C01814=1119.422,-26.499,-49.584,179.647,5.895,149.157
C01815=1119.427,-26.749,-49.572,179.647,5.891,149.156
C01816=1119.432,-26.999,-49.560,179.648,5.887,149.155
C01817=1119.437,-27.248,-49.547,179.648,5.883,149.154
C01818=1119.443,-27.498,-49.535,179.649,5.878,149.153
C01819=1119.448,-27.747,-49.523,179.649,5.874,149.152
C01820=1119.453,-27.997,-49.511,179.649,5.870,149.151
C01821=1119.458,-28.247,-49.498,179.650,5.866,149.150
C01822=1119.463,-28.497,-49.486,179.650,5.862,149.149
C01823=1119.469,-28.746,-49.473,179.651,5.857,149.148
C01824=1119.474,-28.996,-49.461,179.651,5.853,149.147
C01825=1119.479,-29.246,-49.449,179.651,5.850,149.146
C01826=1119.484,-29.495,-49.436,179.652,5.845,149.145
C01827=1119.490,-29.745,-49.424,179.652,5.841,149.144
C01828=1119.495,-29.994,-49.412,179.651,5.837,149.143
C01829=1119.500,-30.244,-49.400,179.652,5.832,149.142
C01830=1119.505,-30.494,-49.387,179.652,5.828,149.141
C01831=1119.511,-30.744,-49.375,179.652,5.824,149.140
C01832=1119.516,-30.993,-49.363,179.652,5.820,149.139
C01833=1119.521,-31.243,-49.351,179.652,5.816,149.138
C01834=1119.526,-31.493,-49.338,179.651,5.811,149.137
C01835=1119.530,-31.742,-49.327,179.652,5.807,149.136
C01836=1119.536,-31.992,-49.314,179.651,5.802,149.135
C01837=1119.541,-32.242,-49.302,179.651,5.798,149.135
C01838=1119.546,-32.491,-49.290,179.651,5.794,149.134
C01839=1119.552,-32.741,-49.278,179.651,5.790,149.133
C01840=1119.556,-32.956,-49.268,179.651,5.786,149.132
C01841=1119.561,-33.171,-49.257,179.650,5.781,149.131
C01842=1119.565,-33.386,-49.247,179.650,5.778,149.130
C01843=1119.570,-33.601,-49.235,179.650,5.774,149.130
C01844=1119.574,-33.816,-49.225,179.650,5.770,149.129
C01845=1119.579,-34.031,-49.215,179.649,5.766,149.128
C01846=1119.583,-34.246,-49.205,179.649,5.762,149.127
C01847=1119.587,-34.462,-49.194,179.648,5.758,149.127
C01848=1119.592,-34.712,-49.183,179.648,5.754,149.126
C01849=1119.598,-34.961,-49.170,179.647,5.749,149.125
C01850=1119.603,-35.211,-49.158,179.647,5.745,149.124
C01851=1119.608,-35.461,-49.146,179.646,5.740,149.123
C01852=1119.613,-35.710,-49.134,179.645,5.735,149.123
C01853=1119.618,-35.960,-49.122,179.645,5.731,149.122
C01854=1119.624,-36.210,-49.110,179.644,5.726,149.121
C01855=1119.629,-36.459,-49.098,179.643,5.722,149.120
C01856=1119.635,-36.708,-49.086,179.643,5.717,149.119
C01857=1119.640,-36.958,-49.075,179.642,5.711,149.118
C01858=1119.645,-37.207,-49.062,179.641,5.707,149.118
C01859=1119.650,-37.457,-49.051,179.640,5.702,149.117
C01860=1119.656,-37.707,-49.039,179.639,5.697,149.116
C01861=1119.660,-37.957,-49.027,179.638,5.692,149.115
C01862=1119.665,-38.206,-49.015,179.637,5.687,149.114
C01863=1119.671,-38.456,-49.003,179.636,5.682,149.114
C01864=1119.676,-38.706,-48.991,179.635,5.677,149.113
C01865=1119.681,-38.955,-48.980,179.635,5.673,149.112
C01866=1119.686,-39.205,-48.968,179.633,5.667,149.111
C01867=1119.691,-39.455,-48.955,179.633,5.663,149.110
C01868=1119.697,-39.705,-48.943,179.631,5.657,149.110
C01869=1119.702,-39.954,-48.932,179.630,5.652,149.109
C01870=1119.708,-40.203,-48.921,179.629,5.646,149.108
C01871=1119.713,-40.453,-48.909,179.628,5.642,149.107
C01872=1119.718,-40.703,-48.897,179.627,5.636,149.106
C01873=1119.723,-40.953,-48.885,179.625,5.631,149.106
C01874=1119.729,-41.203,-48.874,179.624,5.626,149.105
C01875=1119.733,-41.453,-48.862,179.623,5.621,149.104
C01876=1119.738,-41.702,-48.850,179.622,5.615,149.103
C01877=1119.744,-41.951,-48.839,179.621,5.610,149.102
C01878=1119.749,-42.201,-48.827,179.619,5.604,149.102
C01879=1119.755,-42.451,-48.815,179.618,5.598,149.101
C01880=1119.759,-42.700,-48.804,179.616,5.593,149.100
C01881=1119.765,-42.950,-48.792,179.615,5.587,149.099
C01882=1119.770,-43.199,-48.781,179.615,5.583,149.098
C01883=1119.775,-43.449,-48.769,179.615,5.577,149.097
C01884=1119.780,-43.699,-48.758,179.615,5.572,149.096
C01885=1119.785,-43.949,-48.746,179.615,5.568,149.095
C01886=1119.790,-44.198,-48.735,179.615,5.563,149.094
C01887=1119.796,-44.449,-48.723,179.616,5.559,149.093
C01888=1119.802,-44.698,-48.712,179.616,5.554,149.092
C01889=1119.807,-44.948,-48.701,179.615,5.549,149.091
C01890=1119.812,-45.198,-48.689,179.616,5.545,149.090
C01891=1119.817,-45.447,-48.677,179.616,5.539,149.088
C01892=1119.823,-45.696,-48.666,179.617,5.535,149.087
C01893=1119.827,-45.946,-48.655,179.616,5.530,149.086
C01894=1119.833,-46.196,-48.643,179.617,5.526,149.085
C01895=1119.838,-46.446,-48.631,179.617,5.521,149.084
C01896=1119.842,-46.661,-48.622,179.617,5.517,149.083
C01897=1119.847,-46.876,-48.612,179.617,5.513,149.082
C01898=1119.851,-47.091,-48.602,179.617,5.509,149.081
C01899=1119.856,-47.307,-48.592,179.618,5.505,149.080
C01900=1119.861,-47.522,-48.582,179.617,5.500,149.080
C01901=1119.865,-47.737,-48.573,179.617,5.496,149.079
C01902=1119.870,-47.952,-48.563,179.618,5.492,149.078
C01903=1119.874,-48.167,-48.553,179.618,5.489,149.077
C01904=1119.879,-48.417,-48.542,179.618,5.484,149.076
C01905=1119.884,-48.667,-48.530,179.619,5.479,149.075
C01906=1119.890,-48.916,-48.520,179.618,5.474,149.074
C01907=1119.895,-49.166,-48.508,179.619,5.470,149.072
C01908=1119.900,-49.415,-48.496,179.619,5.465,149.071
C01909=1119.906,-49.665,-48.485,179.619,5.461,149.070
C01910=1119.911,-49.915,-48.474,179.619,5.456,149.069
C01911=1119.916,-50.165,-48.463,179.619,5.451,149.068
C01912=1119.921,-50.414,-48.451,179.620,5.446,149.067
C01913=1119.926,-50.663,-48.440,179.619,5.442,149.066
C01914=1119.932,-50.914,-48.429,179.620,5.437,149.065
C01915=1119.937,-51.164,-48.418,179.620,5.432,149.064
C01916=1119.942,-51.412,-48.407,179.620,5.427,149.063
C01917=1119.947,-51.662,-48.395,179.620,5.423,149.062
C01918=1119.952,-51.913,-48.384,179.621,5.418,149.061
C01919=1119.958,-52.162,-48.373,179.621,5.414,149.060
C01920=1119.963,-52.412,-48.361,179.621,5.409,149.058
C01921=1119.968,-52.662,-48.351,179.621,5.404,149.057
C01922=1119.974,-52.911,-48.339,179.621,5.400,149.056
C01923=1119.979,-53.161,-48.328,179.621,5.394,149.055
C01924=1119.984,-53.411,-48.318,179.622,5.390,149.054
C01925=1119.990,-53.660,-48.306,179.622,5.385,149.053
C01926=1119.995,-53.910,-48.295,179.622,5.381,149.052
C01927=1120.000,-54.160,-48.284,179.622,5.376,149.051
C01928=1120.006,-54.409,-48.273,179.622,5.371,149.050
C01929=1120.010,-54.659,-48.261,179.622,5.367,149.049
C01930=1120.015,-54.909,-48.251,179.623,5.362,149.048
C01931=1120.021,-55.158,-48.239,179.623,5.357,149.047
C01932=1120.026,-55.408,-48.228,179.623,5.353,149.046
C01933=1120.031,-55.658,-48.217,179.623,5.347,149.044
C01934=1120.036,-55.907,-48.206,179.623,5.344,149.044
C01935=1120.042,-56.158,-48.195,179.623,5.338,149.042
C01936=1120.047,-56.407,-48.184,179.624,5.334,149.041
C01937=1120.052,-56.656,-48.173,179.624,5.329,149.040
C01938=1120.057,-56.906,-48.163,179.624,5.324,149.039
C01939=1120.063,-57.156,-48.151,179.624,5.320,149.038
C01940=1120.068,-57.406,-48.140,179.624,5.315,149.037
C01941=1120.073,-57.656,-48.129,179.625,5.311,149.036
C01942=1120.078,-57.905,-48.119,179.625,5.306,149.035
C01943=1120.084,-58.155,-48.107,179.625,5.302,149.034
C01944=1120.089,-58.404,-48.096,179.625,5.296,149.033
C01945=1120.094,-58.654,-48.086,179.625,5.291,149.032
C01946=1120.099,-58.904,-48.074,179.625,5.287,149.031
C01947=1120.104,-59.153,-48.064,179.625,5.282,149.029
C01948=1120.110,-59.403,-48.052,179.626,5.278,149.029
C01949=1120.115,-59.653,-48.042,179.626,5.273,149.027
C01950=1120.120,-59.903,-48.031,179.626,5.269,149.026
C01951=1120.125,-60.153,-48.020,179.626,5.264,149.025
C01952=1120.130,-60.368,-48.011,179.626,5.259,149.024
C01953=1120.135,-60.582,-48.001,179.625,5.255,149.024
C01954=1120.139,-60.798,-47.992,179.624,5.251,149.023
C01955=1120.144,-61.013,-47.983,179.623,5.246,149.022
C01956=1120.149,-61.229,-47.973,179.623,5.241,149.021
C01957=1120.152,-61.444,-47.965,179.622,5.237,149.021
C01958=1120.157,-61.659,-47.955,179.622,5.233,149.020
C01959=1120.161,-61.874,-47.945,179.621,5.228,149.019
C01960=1120.167,-62.124,-47.935,179.620,5.223,149.018
C01961=1120.172,-62.374,-47.924,179.620,5.218,149.017
C01962=1120.178,-62.623,-47.913,179.619,5.212,149.016
C01963=1120.183,-62.874,-47.902,179.619,5.208,149.015
C01964=1120.188,-63.123,-47.891,179.618,5.202,149.014
C01965=1120.193,-63.373,-47.881,179.618,5.197,149.013
C01966=1120.199,-63.622,-47.871,179.617,5.191,149.012
C01967=1120.204,-63.872,-47.859,179.617,5.187,149.011
C01968=1120.209,-64.122,-47.849,179.616,5.181,149.010
C01969=1120.214,-64.372,-47.839,179.615,5.176,149.010
C01970=1120.220,-64.621,-47.828,179.615,5.170,149.008
C01971=1120.225,-64.871,-47.817,179.614,5.166,149.007
C01972=1120.230,-65.121,-47.807,179.613,5.160,149.007
C01973=1120.235,-65.371,-47.796,179.613,5.155,149.006
C01974=1120.240,-65.620,-47.785,179.612,5.149,149.004
C01975=1120.245,-65.870,-47.775,179.612,5.145,149.004
C01976=1120.251,-66.119,-47.765,179.611,5.139,149.003
C01977=1120.256,-66.370,-47.754,179.611,5.134,149.001
C01978=1120.262,-66.619,-47.744,179.611,5.129,149.001
C01979=1120.267,-66.868,-47.733,179.610,5.123,148.999
C01980=1120.272,-67.118,-47.722,179.610,5.118,148.998
C01981=1120.278,-67.368,-47.712,179.609,5.113,148.998
C01982=1120.283,-67.618,-47.702,179.609,5.108,148.996
C01983=1120.288,-67.868,-47.691,179.609,5.103,148.995
C01984=1120.293,-68.118,-47.681,179.608,5.097,148.994
C01985=1120.298,-68.367,-47.670,179.608,5.092,148.993
C01986=1120.304,-68.616,-47.660,179.607,5.086,148.992
C01987=1120.309,-68.867,-47.649,179.607,5.081,148.991
C01988=1120.315,-69.116,-47.639,179.607,5.076,148.990
C01989=1120.320,-69.366,-47.629,179.606,5.071,148.989
C01990=1120.325,-69.616,-47.618,179.606,5.066,148.988
C01991=1120.331,-69.866,-47.608,179.607,5.060,148.987
C01992=1120.336,-70.116,-47.597,179.606,5.055,148.986
C01993=1120.341,-70.365,-47.587,179.606,5.050,148.985
C01994=1120.347,-70.615,-47.577,179.605,5.045,148.984
C01995=1120.351,-70.865,-47.567,179.605,5.039,148.983
C01996=1120.357,-71.114,-47.557,179.605,5.034,148.982
C01997=1120.362,-71.364,-47.546,179.605,5.029,148.981
C01998=1120.367,-71.614,-47.536,179.605,5.024,148.979
C01999=1120.373,-71.864,-47.526,179.604,5.018,148.978
C02000=1120.379,-72.113,-47.515,179.604,5.013,148.977
C02001=1120.384,-72.364,-47.505,179.604,5.008,148.976
C02002=1120.389,-72.613,-47.495,179.604,5.002,148.975
C02003=1120.394,-72.862,-47.485,179.604,4.997,148.974
C02004=1120.400,-73.112,-47.475,179.603,4.992,148.973
C02005=1120.405,-73.362,-47.464,179.604,4.987,148.972
C02006=1120.410,-73.612,-47.454,179.604,4.982,148.971
C02007=1120.416,-73.861,-47.444,179.603,4.976,148.970
C02008=1120.420,-74.076,-47.435,179.603,4.972,148.969
C02009=1120.425,-74.292,-47.427,179.603,4.967,148.968
C02010=1120.429,-74.508,-47.418,179.603,4.962,148.967
C02011=1120.434,-74.722,-47.409,179.603,4.958,148.966
C02012=1120.439,-74.939,-47.400,179.603,4.954,148.965
C02013=1120.443,-75.154,-47.392,179.603,4.950,148.964
C02014=1120.448,-75.369,-47.383,179.603,4.945,148.963
C02015=1120.452,-75.584,-47.375,179.603,4.940,148.962
C02016=1120.458,-75.834,-47.365,179.603,4.935,148.961
C02017=1120.463,-76.084,-47.354,179.603,4.929,148.960
C02018=1120.468,-76.333,-47.344,179.603,4.925,148.959
C02019=1120.473,-76.583,-47.334,179.603,4.920,148.957
C02020=1120.479,-76.832,-47.324,179.603,4.914,148.956
C02021=1120.484,-77.083,-47.314,179.603,4.909,148.955
C02022=1120.489,-77.333,-47.305,179.603,4.904,148.954
C02023=1120.495,-77.582,-47.294,179.603,4.899,148.953
C02024=1120.500,-77.832,-47.284,179.603,4.893,148.952
C02025=1120.506,-78.082,-47.275,179.603,4.888,148.950
C02026=1120.510,-78.332,-47.265,179.603,4.883,148.949
C02027=1120.516,-78.581,-47.254,179.603,4.878,148.948
C02028=1120.522,-78.831,-47.244,179.604,4.872,148.947
C02029=1120.527,-79.081,-47.235,179.604,4.867,148.946
C02030=1120.532,-79.330,-47.225,179.604,4.862,148.945
C02031=1120.537,-79.580,-47.215,179.604,4.857,148.943
C02032=1120.542,-79.830,-47.205,179.604,4.852,148.942
C02033=1120.548,-80.080,-47.195,179.604,4.847,148.941
C02034=1120.554,-80.329,-47.185,179.605,4.841,148.940
C02035=1120.559,-80.579,-47.176,179.605,4.836,148.939
C02036=1120.565,-80.829,-47.166,179.605,4.831,148.938
C02037=1120.570,-81.079,-47.156,179.605,4.826,148.936
C02038=1120.574,-81.328,-47.146,179.605,4.821,148.935
C02039=1120.580,-81.578,-47.136,179.605,4.816,148.934
C02040=1120.585,-81.828,-47.127,179.606,4.811,148.933
C02041=1120.591,-82.077,-47.117,179.606,4.806,148.932
C02042=1120.597,-82.327,-47.107,179.606,4.801,148.931
C02043=1120.601,-82.577,-47.097,179.607,4.796,148.929
C02044=1120.607,-82.827,-47.088,179.607,4.791,148.928
C02045=1120.612,-83.077,-47.078,179.607,4.786,148.927
C02046=1120.617,-83.326,-47.068,179.608,4.780,148.926
C02047=1120.622,-83.576,-47.059,179.608,4.775,148.924
C02048=1120.628,-83.826,-47.049,179.608,4.770,148.923
C02049=1120.634,-84.076,-47.039,179.609,4.765,148.922
C02050=1120.639,-84.325,-47.030,179.609,4.760,148.921
C02051=1120.644,-84.575,-47.019,179.609,4.755,148.920
C02052=1120.649,-84.825,-47.010,179.609,4.750,148.919
C02053=1120.655,-85.075,-47.000,179.609,4.745,148.917
C02054=1120.660,-85.324,-46.991,179.611,4.740,148.916
C02055=1120.665,-85.574,-46.981,179.611,4.735,148.915
C02056=1120.670,-85.824,-46.972,179.611,4.730,148.914
C02057=1120.676,-86.073,-46.962,179.611,4.724,148.912
C02058=1120.681,-86.323,-46.953,179.612,4.720,148.911
C02059=1120.687,-86.573,-46.943,179.612,4.715,148.910
C02060=1120.692,-86.823,-46.934,179.612,4.710,148.909
C02061=1120.697,-87.073,-46.923,179.614,4.705,148.907
C02062=1120.702,-87.323,-46.914,179.614,4.700,148.906
C02063=1120.708,-87.572,-46.904,179.614,4.695,148.905
C02064=1120.713,-87.787,-46.896,179.614,4.691,148.904
C02065=1120.717,-88.003,-46.888,179.615,4.686,148.903
C02066=1120.722,-88.218,-46.880,179.615,4.682,148.902
C02067=1120.726,-88.434,-46.872,179.616,4.678,148.901
C02068=1120.730,-88.650,-46.864,179.616,4.673,148.900
C02069=1120.736,-88.865,-46.855,179.617,4.669,148.899
C02070=1120.740,-89.080,-46.847,179.617,4.665,148.898
C02071=1120.745,-89.295,-46.839,179.618,4.661,148.897
C02072=1120.751,-89.545,-46.830,179.618,4.655,148.895
C02073=1120.755,-89.795,-46.820,179.619,4.651,148.894
C02074=1120.760,-90.045,-46.811,179.619,4.646,148.893
C02075=1120.766,-90.295,-46.800,179.620,4.641,148.892
C02076=1120.771,-90.545,-46.792,179.620,4.636,148.890
C02077=1120.777,-90.795,-46.782,179.621,4.632,148.889
C02078=1120.782,-91.044,-46.772,179.621,4.627,148.888
C02079=1120.788,-91.294,-46.763,179.622,4.622,148.887
C02080=1120.793,-91.544,-46.754,179.623,4.617,148.885
C02081=1120.798,-91.793,-46.744,179.624,4.612,148.884
C02082=1120.803,-92.043,-46.735,179.624,4.607,148.883
C02083=1120.809,-92.293,-46.726,179.625,4.603,148.882
C02084=1120.813,-92.543,-46.716,179.625,4.598,148.881
C02085=1120.819,-92.793,-46.707,179.626,4.593,148.879
C02086=1120.825,-93.043,-46.698,179.627,4.589,148.878
C02087=1120.830,-93.292,-46.688,179.627,4.583,148.877
C02088=1120.835,-93.542,-46.679,179.628,4.579,148.876
C02089=1120.840,-93.792,-46.670,179.629,4.573,148.874
C02090=1120.846,-94.041,-46.660,179.629,4.569,148.873
C02091=1120.851,-94.291,-46.651,179.630,4.565,148.872
C02092=1120.856,-94.541,-46.642,179.630,4.560,148.871
C02093=1120.862,-94.791,-46.633,179.630,4.554,148.870
C02094=1120.867,-95.040,-46.623,179.631,4.550,148.868
C02095=1120.872,-95.290,-46.614,179.631,4.545,148.867
C02096=1120.878,-95.540,-46.605,179.632,4.540,148.866
C02097=1120.883,-95.790,-46.595,179.632,4.535,148.865
C02098=1120.889,-96.039,-46.586,179.633,4.530,148.864
C02099=1120.895,-96.289,-46.577,179.633,4.525,148.862
C02100=1120.900,-96.539,-46.568,179.633,4.520,148.862
C02101=1120.905,-96.789,-46.559,179.633,4.515,148.860
C02102=1120.911,-97.038,-46.549,179.634,4.511,148.859
C02103=1120.916,-97.288,-46.540,179.634,4.506,148.858
C02104=1120.921,-97.538,-46.531,179.634,4.500,148.857
C02105=1120.927,-97.788,-46.522,179.634,4.495,148.856
C02106=1120.932,-98.038,-46.513,179.634,4.490,148.854
C02107=1120.937,-98.287,-46.503,179.635,4.486,148.853
C02108=1120.942,-98.537,-46.494,179.635,4.481,148.852
C02109=1120.948,-98.787,-46.485,179.636,4.475,148.851
C02110=1120.953,-99.037,-46.476,179.636,4.470,148.850
C02111=1120.958,-99.287,-46.467,179.636,4.465,148.848
C02112=1120.964,-99.536,-46.458,179.637,4.461,148.847
C02113=1120.970,-99.786,-46.449,179.637,4.456,148.846
C02114=1120.975,-100.035,-46.439,179.637,4.451,148.845
C02115=1120.980,-100.285,-46.430,179.637,4.446,148.844
C02116=1120.985,-100.535,-46.422,179.637,4.441,148.843
C02117=1120.990,-100.785,-46.413,179.638,4.436,148.842
C02118=1120.996,-101.035,-46.403,179.638,4.431,148.840
C02119=1121.001,-101.285,-46.394,179.639,4.426,148.839
C02120=1121.006,-101.500,-46.387,179.639,4.422,148.838
C02121=1121.011,-101.716,-46.379,179.639,4.417,148.837
C02122=1121.015,-101.931,-46.371,179.639,4.413,148.836
C02123=1121.020,-102.146,-46.363,179.640,4.409,148.835
C02124=1121.025,-102.363,-46.356,179.639,4.404,148.834
C02125=1121.029,-102.578,-46.349,179.640,4.400,148.833
C02126=1121.034,-102.793,-46.341,179.641,4.396,148.832
C02127=1121.039,-103.009,-46.332,179.640,4.391,148.831
C02128=1121.044,-103.259,-46.323,179.640,4.386,148.830
C02129=1121.050,-103.509,-46.315,179.641,4.381,148.829
C02130=1121.055,-103.758,-46.306,179.642,4.376,148.827
C02131=1121.060,-104.008,-46.297,179.642,4.371,148.826
C02132=1121.065,-104.258,-46.288,179.642,4.366,148.825
C02133=1121.071,-104.507,-46.279,179.642,4.361,148.824
C02134=1121.076,-104.757,-46.270,179.642,4.355,148.823
C02135=1121.082,-105.007,-46.261,179.643,4.350,148.822
C02136=1121.087,-105.257,-46.252,179.643,4.345,148.820
C02137=1121.092,-105.507,-46.243,179.643,4.340,148.819
C02138=1121.098,-105.756,-46.235,179.643,4.336,148.818
C02139=1121.103,-106.006,-46.226,179.644,4.331,148.817
C02140=1121.108,-106.256,-46.217,179.644,4.326,148.816
C02141=1121.114,-106.506,-46.208,179.644,4.321,148.815
C02142=1121.119,-106.755,-46.199,179.644,4.315,148.813
C02143=1121.125,-107.005,-46.191,179.645,4.310,148.812
C02144=1121.130,-107.255,-46.182,179.645,4.305,148.811
C02145=1121.135,-107.505,-46.173,179.645,4.300,148.810
C02146=1121.140,-107.755,-46.164,179.645,4.295,148.809
C02147=1121.145,-108.005,-46.156,179.646,4.290,148.807
C02148=1121.151,-108.254,-46.147,179.646,4.284,148.806
C02149=1121.157,-108.504,-46.138,179.646,4.279,148.805
C02150=1121.162,-108.754,-46.129,179.646,4.274,148.804
C02151=1121.168,-109.004,-46.120,179.647,4.269,148.803
C02152=1121.173,-109.253,-46.112,179.647,4.264,148.801
C02153=1121.179,-109.503,-46.103,179.647,4.258,148.800
C02154=1121.184,-109.753,-46.094,179.647,4.253,148.799
C02155=1121.189,-110.003,-46.085,179.648,4.248,148.798
C02156=1121.195,-110.253,-46.077,179.648,4.243,148.797
C02157=1121.200,-110.503,-46.069,179.648,4.238,148.795
C02158=1121.205,-110.752,-46.060,179.648,4.233,148.794
C02159=1121.211,-111.002,-46.051,179.649,4.227,148.793
C02160=1121.216,-111.251,-46.042,179.649,4.222,148.792
C02161=1121.221,-111.502,-46.035,179.649,4.217,148.791
C02162=1121.226,-111.751,-46.026,179.649,4.212,148.789
C02163=1121.232,-112.001,-46.017,179.650,4.207,148.788
C02164=1121.237,-112.251,-46.009,179.649,4.202,148.787
C02165=1121.243,-112.501,-46.000,179.650,4.197,148.786
C02166=1121.248,-112.750,-45.992,179.650,4.192,148.785
C02167=1121.254,-113.000,-45.983,179.650,4.186,148.784
C02168=1121.259,-113.250,-45.975,179.650,4.181,148.782
C02169=1121.264,-113.500,-45.966,179.651,4.176,148.781
C02170=1121.270,-113.749,-45.957,179.651,4.171,148.780
C02171=1121.275,-114.000,-45.949,179.652,4.165,148.779
C02172=1121.281,-114.250,-45.940,179.652,4.160,148.777
C02173=1121.286,-114.499,-45.931,179.652,4.155,148.776
C02174=1121.292,-114.749,-45.923,179.653,4.150,148.775
C02175=1121.296,-114.999,-45.915,179.653,4.145,148.774
C02176=1121.301,-115.215,-45.908,179.653,4.140,148.773
C02177=1121.306,-115.430,-45.900,179.653,4.136,148.772
C02178=1121.311,-115.645,-45.894,179.653,4.131,148.771
C02179=1121.316,-115.861,-45.886,179.653,4.127,148.770
C02180=1121.321,-116.077,-45.879,179.653,4.122,148.769
C02181=1121.325,-116.292,-45.872,179.654,4.118,148.768
C02182=1121.329,-116.508,-45.864,179.654,4.113,148.767
C02183=1121.334,-116.723,-45.857,179.654,4.108,148.766
C02184=1121.340,-116.974,-45.849,179.654,4.103,148.764
C02185=1121.345,-117.223,-45.840,179.654,4.098,148.763
C02186=1121.351,-117.473,-45.832,179.655,4.092,148.762
C02187=1121.356,-117.722,-45.824,179.655,4.087,148.761
C02188=1121.361,-117.973,-45.816,179.655,4.082,148.759
C02189=1121.366,-118.223,-45.807,179.656,4.077,148.758
C02190=1121.373,-118.472,-45.799,179.655,4.071,148.757
C02191=1121.378,-118.722,-45.790,179.656,4.066,148.756
C02192=1121.383,-118.972,-45.783,179.656,4.060,148.755
C02193=1121.388,-119.221,-45.774,179.656,4.055,148.753
C02194=1121.394,-119.472,-45.766,179.657,4.050,148.752
C02195=1121.399,-119.721,-45.757,179.657,4.045,148.751
C02196=1121.405,-119.972,-45.749,179.657,4.039,148.750
C02197=1121.410,-120.220,-45.741,179.657,4.034,148.748
C02198=1121.415,-120.471,-45.733,179.658,4.028,148.747
C02199=1121.421,-120.720,-45.725,179.658,4.023,148.746
C02200=1121.427,-120.970,-45.716,179.658,4.018,148.745
C02201=1121.431,-121.220,-45.708,179.658,4.012,148.743
C02202=1121.437,-121.470,-45.700,179.658,4.007,148.742
C02203=1121.443,-121.720,-45.692,179.658,4.001,148.741
C02204=1121.448,-121.969,-45.684,179.659,3.996,148.740
C02205=1121.453,-122.220,-45.676,179.658,3.990,148.739
C02206=1121.459,-122.469,-45.667,179.659,3.985,148.737
C02207=1121.464,-122.719,-45.659,179.660,3.979,148.736
C02208=1121.470,-122.969,-45.652,179.660,3.974,148.735
C02209=1121.475,-123.218,-45.643,179.660,3.968,148.733
C02210=1121.481,-123.468,-45.635,179.660,3.963,148.732
C02211=1121.486,-123.718,-45.628,179.660,3.958,148.731
C02212=1121.491,-123.968,-45.619,179.660,3.953,148.730
C02213=1121.497,-124.218,-45.611,179.661,3.946,148.728
C02214=1121.502,-124.467,-45.604,179.661,3.941,148.727
C02215=1121.507,-124.717,-45.595,179.661,3.936,148.726
C02216=1121.513,-124.967,-45.588,179.661,3.930,148.725
C02217=1121.518,-125.217,-45.579,179.661,3.925,148.724
C02218=1121.524,-125.467,-45.572,179.662,3.919,148.722
C02219=1121.529,-125.717,-45.563,179.662,3.913,148.721
C02220=1121.535,-125.966,-45.555,179.662,3.908,148.720
C02221=1121.540,-126.217,-45.547,179.662,3.903,148.718
C02222=1121.546,-126.466,-45.540,179.662,3.897,148.717
C02223=1121.551,-126.716,-45.531,179.663,3.891,148.716
C02224=1121.556,-126.966,-45.524,179.663,3.886,148.715
C02225=1121.562,-127.215,-45.516,179.663,3.880,148.713
C02226=1121.567,-127.466,-45.509,179.663,3.875,148.712
C02227=1121.573,-127.715,-45.500,179.664,3.870,148.711
C02228=1121.578,-127.965,-45.492,179.664,3.864,148.709
C02229=1121.583,-128.215,-45.485,179.664,3.858,148.708
C02230=1121.589,-128.465,-45.476,179.664,3.852,148.707
C02231=1121.594,-128.715,-45.469,179.665,3.847,148.706
C02232=1121.171,-128.705,-45.495,179.672,3.851,148.704
C02233=1121.166,-128.455,-45.502,179.672,3.857,148.706
C02234=1121.161,-128.205,-45.511,179.672,3.863,148.707
C02235=1121.155,-127.956,-45.519,179.671,3.868,148.708
C02236=1121.150,-127.705,-45.526,179.671,3.873,148.709
C02237=1121.144,-127.456,-45.534,179.671,3.879,148.711
C02238=1121.139,-127.206,-45.541,179.671,3.884,148.712
C02239=1121.133,-126.956,-45.550,179.670,3.890,148.713
C02240=1121.127,-126.707,-45.558,179.670,3.896,148.715
C02241=1121.123,-126.456,-45.566,179.670,3.901,148.716
C02242=1121.117,-126.207,-45.573,179.670,3.906,148.717
C02243=1121.112,-125.957,-45.582,179.669,3.913,148.718
C02244=1121.106,-125.707,-45.590,179.669,3.918,148.720
C02245=1121.101,-125.457,-45.598,179.669,3.923,148.721
C02246=1121.096,-125.208,-45.606,179.669,3.929,148.722
C02247=1121.090,-124.958,-45.614,179.669,3.934,148.723
C02248=1121.084,-124.708,-45.622,179.668,3.940,148.725
C02249=1121.080,-124.458,-45.630,179.668,3.946,148.726
C02250=1121.074,-124.208,-45.638,179.668,3.951,148.727
C02251=1121.068,-123.958,-45.646,179.668,3.956,148.728
C02252=1121.063,-123.709,-45.654,179.667,3.961,148.730
C02253=1121.058,-123.459,-45.662,179.667,3.968,148.731
C02254=1121.051,-123.209,-45.670,179.667,3.973,148.732
C02255=1121.047,-122.959,-45.678,179.666,3.978,148.733
C02256=1121.041,-122.710,-45.686,179.666,3.983,148.735
C02257=1121.035,-122.459,-45.694,179.666,3.989,148.736
C02258=1121.030,-122.210,-45.703,179.666,3.994,148.737
C02259=1121.025,-121.960,-45.710,179.665,4.000,148.739
C02260=1121.020,-121.710,-45.719,179.665,4.005,148.740
C02261=1121.014,-121.460,-45.727,179.665,4.011,148.741
C02262=1121.009,-121.211,-45.735,179.665,4.016,148.742
C02263=1121.003,-120.961,-45.743,179.665,4.022,148.743
C02264=1120.998,-120.711,-45.752,179.665,4.027,148.745
C02265=1120.992,-120.461,-45.760,179.664,4.032,148.746
C02266=1120.987,-120.211,-45.768,179.665,4.038,148.747
C02267=1120.982,-119.961,-45.776,179.664,4.043,148.748
C02268=1120.976,-119.712,-45.784,179.663,4.049,148.750
C02269=1120.971,-119.462,-45.793,179.663,4.054,148.751
C02270=1120.965,-119.212,-45.801,179.663,4.059,148.752
C02271=1120.960,-118.962,-45.809,179.663,4.064,148.753
C02272=1120.955,-118.713,-45.818,179.663,4.070,148.754
C02273=1120.949,-118.463,-45.826,179.663,4.075,148.756
C02274=1120.944,-118.213,-45.835,179.662,4.080,148.757
C02275=1120.938,-117.963,-45.843,179.662,4.086,148.758
C02276=1120.933,-117.714,-45.851,179.662,4.091,148.759
C02277=1120.928,-117.463,-45.859,179.662,4.096,148.761
C02278=1120.922,-117.214,-45.868,179.661,4.101,148.762
C02279=1120.917,-116.963,-45.876,179.662,4.107,148.763
C02280=1120.911,-116.714,-45.884,179.661,4.113,148.764
C02281=1120.907,-116.499,-45.892,179.660,4.117,148.765
C02282=1120.902,-116.283,-45.899,179.661,4.121,148.766
C02283=1120.898,-116.068,-45.906,179.660,4.126,148.767
C02284=1120.893,-115.852,-45.914,179.660,4.131,148.768
C02285=1120.888,-115.637,-45.921,179.660,4.135,148.769
C02286=1120.883,-115.421,-45.928,179.660,4.140,148.771
C02287=1120.879,-115.205,-45.936,179.659,4.144,148.772
C02288=1120.874,-114.989,-45.943,179.659,4.149,148.773
C02289=1120.869,-114.739,-45.952,179.659,4.154,148.774
C02290=1120.863,-114.490,-45.959,179.659,4.159,148.775
C02291=1120.858,-114.240,-45.968,179.659,4.164,148.776
C02292=1120.853,-113.990,-45.977,179.658,4.169,148.777
C02293=1120.847,-113.740,-45.985,179.658,4.174,148.779
C02294=1120.842,-113.491,-45.994,179.658,4.180,148.780
C02295=1120.837,-113.241,-46.003,179.658,4.185,148.781
C02296=1120.831,-112.992,-46.011,179.657,4.190,148.782
C02297=1120.825,-112.741,-46.019,179.658,4.196,148.783
C02298=1120.820,-112.491,-46.028,179.657,4.201,148.785
C02299=1120.815,-112.241,-46.037,179.657,4.206,148.786
C02300=1120.809,-111.992,-46.046,179.657,4.211,148.787
C02301=1120.804,-111.742,-46.054,179.657,4.217,148.788
C02302=1120.799,-111.492,-46.063,179.656,4.222,148.789
C02303=1120.793,-111.243,-46.071,179.656,4.227,148.791
C02304=1120.788,-110.993,-46.080,179.656,4.232,148.792
C02305=1120.782,-110.743,-46.088,179.656,4.237,148.793
C02306=1120.777,-110.493,-46.097,179.655,4.242,148.794
C02307=1120.771,-110.244,-46.106,179.655,4.248,148.795
C02308=1120.766,-109.994,-46.115,179.655,4.253,148.797
C02309=1120.761,-109.744,-46.123,179.655,4.258,148.798
C02310=1120.756,-109.494,-46.132,179.654,4.263,148.799
C02311=1120.750,-109.244,-46.140,179.654,4.268,148.800
C02312=1120.744,-108.994,-46.149,179.653,4.273,148.801
C02313=1120.739,-108.744,-46.158,179.653,4.278,148.803
C02314=1120.734,-108.495,-46.167,179.653,4.283,148.804
C02315=1120.728,-108.246,-46.175,179.653,4.288,148.805
C02316=1120.723,-107.996,-46.184,179.652,4.293,148.806
C02317=1120.718,-107.746,-46.193,179.652,4.298,148.807
C02318=1120.713,-107.496,-46.202,179.652,4.304,148.809
C02319=1120.707,-107.245,-46.210,179.652,4.309,148.810
C02320=1120.702,-106.996,-46.219,179.651,4.314,148.811
C02321=1120.696,-106.746,-46.228,179.651,4.319,148.812
C02322=1120.691,-106.496,-46.237,179.651,4.324,148.813
C02323=1120.685,-106.246,-46.246,179.651,4.329,148.815
C02324=1120.680,-105.997,-46.255,179.650,4.335,148.816
C02325=1120.674,-105.747,-46.264,179.650,4.340,148.817
C02326=1120.669,-105.498,-46.272,179.650,4.345,148.818
C02327=1120.664,-105.248,-46.281,179.649,4.349,148.819
C02328=1120.659,-104.998,-46.290,179.649,4.354,148.821
C02329=1120.654,-104.748,-46.299,179.649,4.359,148.821
C02330=1120.648,-104.498,-46.309,179.649,4.364,148.823
C02331=1120.642,-104.249,-46.317,179.649,4.370,148.824
C02332=1120.637,-103.999,-46.326,179.648,4.375,148.825
C02333=1120.632,-103.749,-46.335,179.648,4.380,148.826
C02334=1120.627,-103.499,-46.344,179.648,4.385,148.827
C02335=1120.621,-103.249,-46.353,179.647,4.389,148.829
C02336=1120.616,-102.999,-46.362,179.647,4.395,148.830
C02337=1120.611,-102.784,-46.369,179.647,4.399,148.831
C02338=1120.607,-102.568,-46.378,179.646,4.404,148.832
C02339=1120.602,-102.353,-46.385,179.646,4.408,148.833
C02340=1120.598,-102.137,-46.393,179.646,4.413,148.834
C02341=1120.593,-101.922,-46.401,179.646,4.416,148.835
C02342=1120.588,-101.706,-46.409,179.645,4.421,148.836
C02343=1120.584,-101.491,-46.417,179.646,4.426,148.837
C02344=1120.579,-101.276,-46.424,179.645,4.430,148.838
C02345=1120.574,-101.026,-46.433,179.645,4.435,148.839
C02346=1120.568,-100.776,-46.443,179.645,4.440,148.840
C02347=1120.563,-100.526,-46.452,179.644,4.444,148.841
C02348=1120.557,-100.277,-46.460,179.644,4.449,148.843
C02349=1120.552,-100.027,-46.469,179.644,4.455,148.844
C02350=1120.547,-99.777,-46.478,179.643,4.460,148.845
C02351=1120.541,-99.527,-46.488,179.643,4.465,148.846
C02352=1120.536,-99.277,-46.497,179.642,4.469,148.847
C02353=1120.531,-99.028,-46.506,179.643,4.474,148.848
C02354=1120.525,-98.777,-46.516,179.642,4.479,148.850
C02355=1120.520,-98.528,-46.524,179.642,4.484,148.851
C02356=1120.514,-98.278,-46.533,179.642,4.490,148.852
C02357=1120.509,-98.029,-46.542,179.641,4.494,148.853
C02358=1120.504,-97.779,-46.552,179.641,4.499,148.854
C02359=1120.498,-97.529,-46.561,179.641,4.504,148.856
C02360=1120.493,-97.279,-46.570,179.640,4.509,148.857
C02361=1120.487,-97.029,-46.580,179.640,4.515,148.858
C02362=1120.482,-96.780,-46.589,179.639,4.519,148.859
C02363=1120.477,-96.530,-46.598,179.639,4.524,148.860
C02364=1120.471,-96.280,-46.608,179.639,4.529,148.861
C02365=1120.466,-96.030,-46.616,179.639,4.534,148.863
C02366=1120.461,-95.781,-46.626,179.638,4.539,148.864
C02367=1120.455,-95.531,-46.636,179.638,4.544,148.865
C02368=1120.450,-95.281,-46.644,179.638,4.549,148.866
C02369=1120.445,-95.031,-46.653,179.638,4.554,148.867
C02370=1120.440,-94.781,-46.664,179.637,4.558,148.868
C02371=1120.434,-94.532,-46.672,179.637,4.563,148.870
C02372=1120.429,-94.282,-46.681,179.637,4.569,148.871
C02373=1120.424,-94.032,-46.692,179.636,4.573,148.872
C02374=1120.418,-93.782,-46.700,179.635,4.578,148.873
C02375=1120.413,-93.532,-46.710,179.634,4.583,148.875
C02376=1120.408,-93.283,-46.720,179.634,4.587,148.876
C02377=1120.403,-93.033,-46.728,179.633,4.592,148.877
C02378=1120.397,-92.783,-46.738,179.632,4.597,148.878
C02379=1120.392,-92.534,-46.748,179.631,4.601,148.879
C02380=1120.387,-92.284,-46.756,179.631,4.607,148.881
C02381=1120.381,-92.034,-46.766,179.630,4.611,148.882
C02382=1120.376,-91.784,-46.776,179.630,4.616,148.883
C02383=1120.370,-91.534,-46.785,179.629,4.621,148.884
C02384=1120.365,-91.285,-46.795,179.629,4.626,148.886
C02385=1120.359,-91.035,-46.804,179.628,4.630,148.887
C02386=1120.354,-90.785,-46.813,179.628,4.635,148.888
C02387=1120.349,-90.536,-46.823,179.627,4.640,148.889
C02388=1120.343,-90.286,-46.832,179.626,4.645,148.891
C02389=1120.338,-90.036,-46.842,179.625,4.650,148.892
C02390=1120.332,-89.786,-46.851,179.625,4.655,148.893
C02391=1120.327,-89.536,-46.860,179.625,4.660,148.894
C02392=1120.322,-89.287,-46.870,179.624,4.664,148.895
C02393=1120.317,-89.071,-46.878,179.624,4.669,148.897
C02394=1120.313,-88.856,-46.886,179.623,4.673,148.897
C02395=1120.308,-88.640,-46.895,179.622,4.677,148.899
C02396=1120.304,-88.425,-46.903,179.623,4.682,148.900
C02397=1120.299,-88.210,-46.911,179.622,4.686,148.901
C02398=1120.295,-87.994,-46.920,179.622,4.690,148.902
C02399=1120.290,-87.779,-46.928,179.621,4.695,148.903
C02400=1120.285,-87.563,-46.936,179.621,4.698,148.904
C02401=1120.280,-87.314,-46.946,179.621,4.704,148.905
C02402=1120.275,-87.064,-46.955,179.620,4.709,148.906
C02403=1120.269,-86.814,-46.965,179.619,4.714,148.908
C02404=1120.264,-86.564,-46.974,179.619,4.719,148.909
C02405=1120.258,-86.315,-46.984,179.619,4.724,148.910
C02406=1120.254,-86.064,-46.993,179.619,4.729,148.911
C02407=1120.248,-85.815,-47.004,179.618,4.733,148.912
C02408=1120.243,-85.566,-47.013,179.618,4.739,148.914
C02409=1120.237,-85.315,-47.023,179.617,4.744,148.915
C02410=1120.232,-85.066,-47.032,179.617,4.749,148.916
C02411=1120.227,-84.816,-47.042,179.616,4.754,148.917
C02412=1120.222,-84.567,-47.051,179.616,4.759,148.918
C02413=1120.216,-84.317,-47.061,179.616,4.764,148.920
C02414=1120.211,-84.067,-47.071,179.615,4.769,148.921
C02415=1120.206,-83.817,-47.081,179.615,4.774,148.922
C02416=1120.200,-83.567,-47.091,179.614,4.779,148.923
C02417=1120.195,-83.318,-47.100,179.614,4.784,148.925
C02418=1120.189,-83.068,-47.110,179.614,4.789,148.926
C02419=1120.184,-82.818,-47.119,179.613,4.794,148.927
C02420=1120.179,-82.569,-47.130,179.613,4.800,148.928
C02421=1120.173,-82.318,-47.139,179.613,4.805,148.929
C02422=1120.169,-82.069,-47.149,179.613,4.810,148.930
C02423=1120.163,-81.819,-47.159,179.613,4.815,148.932
C02424=1120.158,-81.569,-47.168,179.613,4.820,148.933
C02425=1120.152,-81.320,-47.178,179.612,4.825,148.934
C02426=1120.147,-81.070,-47.189,179.612,4.830,148.935
C02427=1120.142,-80.820,-47.198,179.612,4.835,148.936
C02428=1120.136,-80.570,-47.208,179.611,4.840,148.937
C02429=1120.131,-80.321,-47.218,179.611,4.845,148.939
C02430=1120.126,-80.071,-47.228,179.611,4.850,148.940
C02431=1120.120,-79.821,-47.237,179.611,4.855,148.941
C02432=1120.115,-79.571,-47.248,179.611,4.861,148.942
C02433=1120.110,-79.322,-47.258,179.611,4.866,148.943
C02434=1120.104,-79.072,-47.267,179.610,4.871,148.945
C02435=1120.099,-78.822,-47.277,179.610,4.876,148.946
C02436=1120.093,-78.572,-47.287,179.610,4.881,148.947
C02437=1120.089,-78.323,-47.297,179.610,4.886,148.948
C02438=1120.083,-78.073,-47.308,179.610,4.892,148.949
C02439=1120.077,-77.823,-47.317,179.610,4.898,148.950
C02440=1120.073,-77.574,-47.327,179.610,4.903,148.952
C02441=1120.067,-77.324,-47.337,179.610,4.908,148.953
C02442=1120.062,-77.074,-47.348,179.610,4.913,148.954
C02443=1120.056,-76.824,-47.358,179.610,4.918,148.955
C02444=1120.051,-76.574,-47.367,179.609,4.923,148.956
C02445=1120.046,-76.325,-47.377,179.609,4.928,148.957
C02446=1120.041,-76.075,-47.387,179.609,4.934,148.959
C02447=1120.035,-75.825,-47.398,179.609,4.938,148.959
C02448=1120.029,-75.576,-47.408,179.610,4.944,148.961
C02449=1120.025,-75.360,-47.417,179.609,4.949,148.962
C02450=1120.021,-75.144,-47.425,179.610,4.953,148.963
C02451=1120.016,-74.930,-47.433,179.609,4.957,148.964
C02452=1120.011,-74.714,-47.443,179.610,4.962,148.965
C02453=1120.007,-74.498,-47.451,179.610,4.967,148.965
C02454=1120.002,-74.284,-47.460,179.610,4.971,148.966
C02455=1119.998,-74.069,-47.468,179.610,4.976,148.968
C02456=1119.993,-73.853,-47.478,179.609,4.980,148.969
C02457=1119.988,-73.603,-47.488,179.610,4.986,148.969
C02458=1119.983,-73.353,-47.498,179.610,4.991,148.971
C02459=1119.977,-73.104,-47.509,179.610,4.996,148.972
C02460=1119.972,-72.854,-47.518,179.610,5.001,148.973
C02461=1119.966,-72.604,-47.528,179.610,5.006,148.974
C02462=1119.961,-72.354,-47.538,179.611,5.012,148.975
C02463=1119.956,-72.104,-47.549,179.611,5.017,148.976
C02464=1119.950,-71.855,-47.559,179.610,5.022,148.977
C02465=1119.945,-71.605,-47.570,179.611,5.028,148.978
C02466=1119.940,-71.356,-47.580,179.611,5.033,148.979
C02467=1119.934,-71.106,-47.590,179.611,5.038,148.981
C02468=1119.930,-70.856,-47.600,179.612,5.043,148.982
C02469=1119.924,-70.607,-47.611,179.612,5.049,148.983
C02470=1119.919,-70.357,-47.621,179.612,5.053,148.984
C02471=1119.914,-70.107,-47.631,179.612,5.059,148.985
C02472=1119.908,-69.857,-47.642,179.613,5.065,148.986
C02473=1119.903,-69.607,-47.652,179.613,5.069,148.987
C02474=1119.898,-69.358,-47.662,179.613,5.074,148.988
C02475=1119.892,-69.108,-47.673,179.614,5.080,148.989
C02476=1119.887,-68.858,-47.683,179.614,5.085,148.990
C02477=1119.881,-68.608,-47.693,179.614,5.090,148.991
C02478=1119.877,-68.359,-47.705,179.615,5.096,148.992
C02479=1119.871,-68.109,-47.715,179.615,5.101,148.993
C02480=1119.866,-67.860,-47.725,179.615,5.106,148.994
C02481=1119.861,-67.609,-47.736,179.616,5.111,148.995
C02482=1119.855,-67.360,-47.746,179.616,5.116,148.996
C02483=1119.850,-67.110,-47.757,179.617,5.122,148.997
C02484=1119.845,-66.861,-47.767,179.617,5.127,148.998
C02485=1119.840,-66.610,-47.778,179.617,5.132,148.999
C02486=1119.834,-66.361,-47.788,179.617,5.138,149.000
C02487=1119.828,-66.111,-47.798,179.618,5.143,149.001
C02488=1119.824,-65.862,-47.810,179.619,5.148,149.002
C02489=1119.818,-65.612,-47.820,179.619,5.153,149.003
C02490=1119.813,-65.362,-47.830,179.619,5.158,149.004
C02491=1119.808,-65.112,-47.841,179.620,5.164,149.005
C02492=1119.803,-64.863,-47.852,179.620,5.169,149.006
C02493=1119.797,-64.613,-47.862,179.621,5.174,149.007
C02494=1119.792,-64.363,-47.873,179.621,5.179,149.008
C02495=1119.787,-64.114,-47.884,179.622,5.185,149.009
C02496=1119.782,-63.864,-47.894,179.622,5.190,149.010
C02497=1119.776,-63.614,-47.904,179.623,5.195,149.011
C02498=1119.771,-63.364,-47.916,179.623,5.200,149.012
C02499=1119.765,-63.115,-47.927,179.624,5.206,149.013
C02500=1119.760,-62.865,-47.937,179.625,5.211,149.014
C02501=1119.755,-62.616,-47.948,179.626,5.216,149.015
C02502=1119.750,-62.365,-47.959,179.626,5.221,149.016
C02503=1119.745,-62.116,-47.970,179.627,5.227,149.017
C02504=1119.740,-61.866,-47.980,179.627,5.232,149.018
C02505=1119.735,-61.651,-47.989,179.628,5.236,149.019
C02506=1119.731,-61.435,-47.999,179.628,5.241,149.020
C02507=1119.726,-61.220,-48.009,179.629,5.245,149.020
C02508=1119.722,-61.005,-48.018,179.630,5.250,149.021
C02509=1119.717,-60.789,-48.027,179.630,5.254,149.022
C02510=1119.712,-60.575,-48.036,179.631,5.259,149.023
C02511=1119.708,-60.360,-48.046,179.632,5.263,149.023
C02512=1119.703,-60.145,-48.055,179.632,5.267,149.024
C02513=1119.698,-59.895,-48.067,179.632,5.272,149.025
C02514=1119.692,-59.645,-48.077,179.632,5.277,149.026
C02515=1119.688,-59.395,-48.088,179.632,5.281,149.027
C02516=1119.683,-59.145,-48.099,179.632,5.286,149.029
C02517=1119.677,-58.896,-48.110,179.631,5.290,149.029
C02518=1119.672,-58.646,-48.121,179.631,5.295,149.031
C02519=1119.666,-58.397,-48.132,179.631,5.300,149.032
C02520=1119.661,-58.147,-48.142,179.631,5.304,149.033
C02521=1119.657,-57.897,-48.154,179.631,5.310,149.034
C02522=1119.650,-57.647,-48.165,179.630,5.314,149.035
C02523=1119.646,-57.397,-48.176,179.631,5.319,149.036
C02524=1119.641,-57.148,-48.187,179.630,5.323,149.037
C02525=1119.635,-56.898,-48.197,179.630,5.328,149.038
C02526=1119.630,-56.648,-48.209,179.630,5.333,149.039
C02527=1119.624,-56.399,-48.219,179.629,5.337,149.040
C02528=1119.620,-56.149,-48.231,179.630,5.342,149.041
C02529=1119.615,-55.900,-48.242,179.629,5.346,149.042
C02530=1119.609,-55.650,-48.253,179.629,5.352,149.043
C02531=1119.604,-55.400,-48.264,179.629,5.356,149.044
C02532=1119.599,-55.150,-48.275,179.629,5.361,149.046
C02533=1119.593,-54.901,-48.286,179.629,5.366,149.047
C02534=1119.588,-54.651,-48.297,179.629,5.370,149.048
C02535=1119.583,-54.401,-48.308,179.628,5.375,149.049
C02536=1119.577,-54.151,-48.320,179.628,5.379,149.050
C02537=1119.572,-53.902,-48.331,179.628,5.384,149.051
C02538=1119.568,-53.652,-48.342,179.628,5.389,149.052
C02539=1119.561,-53.402,-48.353,179.627,5.393,149.053
C02540=1119.557,-53.153,-48.364,179.628,5.398,149.054
C02541=1119.552,-52.903,-48.376,179.627,5.403,149.055
C02542=1119.546,-52.653,-48.386,179.627,5.408,149.056
C02543=1119.541,-52.404,-48.398,179.627,5.412,149.057
C02544=1119.536,-52.154,-48.409,179.627,5.417,149.058
C02545=1119.530,-51.905,-48.420,179.627,5.422,149.060
C02546=1119.525,-51.654,-48.431,179.626,5.426,149.061
C02547=1119.520,-51.405,-48.443,179.626,5.431,149.062
C02548=1119.515,-51.155,-48.454,179.626,5.436,149.063
C02549=1119.509,-50.906,-48.466,179.626,5.440,149.064
C02550=1119.504,-50.655,-48.476,179.626,5.445,149.065
C02551=1119.499,-50.406,-48.488,179.625,5.450,149.066
C02552=1119.493,-50.157,-48.499,179.625,5.455,149.067
C02553=1119.489,-49.907,-48.510,179.626,5.459,149.068
C02554=1119.483,-49.657,-48.522,179.625,5.464,149.069
C02555=1119.478,-49.407,-48.533,179.625,5.469,149.070
C02556=1119.472,-49.158,-48.544,179.624,5.473,149.071
C02557=1119.468,-48.908,-48.556,179.625,5.478,149.072
C02558=1119.463,-48.658,-48.567,179.624,5.482,149.074
C02559=1119.457,-48.408,-48.579,179.624,5.487,149.075
C02560=1119.452,-48.159,-48.590,179.624,5.492,149.076
C02561=1119.447,-47.944,-48.600,179.624,5.496,149.077
C02562=1119.442,-47.729,-48.610,179.624,5.500,149.077
C02563=1119.438,-47.513,-48.619,179.623,5.504,149.079
C02564=1119.433,-47.298,-48.629,179.623,5.508,149.080
C02565=1119.429,-47.084,-48.639,179.623,5.512,149.080
C02566=1119.425,-46.867,-48.649,179.623,5.516,149.081
C02567=1119.421,-46.652,-48.659,179.623,5.520,149.082
C02568=1119.416,-46.438,-48.669,179.623,5.524,149.083
C02569=1119.410,-46.188,-48.680,179.622,5.529,149.084
C02570=1119.406,-45.939,-48.691,179.623,5.534,149.085
C02571=1119.400,-45.688,-48.703,179.622,5.538,149.086
C02572=1119.395,-45.439,-48.714,179.622,5.544,149.088
C02573=1119.390,-45.189,-48.726,179.621,5.548,149.089
C02574=1119.385,-44.940,-48.737,179.622,5.553,149.090
C02575=1119.379,-44.690,-48.749,179.622,5.558,149.091
C02576=1119.374,-44.440,-48.760,179.621,5.562,149.092
C02577=1119.369,-44.190,-48.772,179.622,5.567,149.093
C02578=1119.364,-43.940,-48.784,179.621,5.571,149.094
C02579=1119.358,-43.691,-48.795,179.621,5.576,149.095
C02580=1119.353,-43.441,-48.806,179.621,5.581,149.096
C02581=1119.348,-43.192,-48.818,179.621,5.585,149.097
C02582=1119.343,-42.942,-48.830,179.621,5.591,149.098
C02583=1119.338,-42.692,-48.841,179.623,5.597,149.099
C02584=1119.332,-42.443,-48.852,179.624,5.602,149.100
C02585=1119.327,-42.193,-48.864,179.625,5.608,149.101
C02586=1119.322,-41.943,-48.876,179.626,5.613,149.101
C02587=1119.316,-41.693,-48.887,179.627,5.618,149.102
C02588=1119.311,-41.444,-48.899,179.629,5.623,149.103
C02589=1119.307,-41.195,-48.911,179.630,5.629,149.104
C02590=1119.301,-40.945,-48.923,179.631,5.634,149.105
C02591=1119.296,-40.695,-48.935,179.633,5.640,149.105
C02592=1119.290,-40.446,-48.946,179.634,5.645,149.106
C02593=1119.285,-40.196,-48.958,179.635,5.650,149.107
C02594=1119.280,-39.946,-48.970,179.636,5.655,149.108
C02595=1119.275,-39.696,-48.981,179.637,5.660,149.109
C02596=1119.270,-39.447,-48.994,179.638,5.666,149.109
C02597=1119.264,-39.197,-49.006,179.639,5.670,149.110
C02598=1119.260,-38.947,-49.017,179.640,5.676,149.111
C02599=1119.254,-38.697,-49.029,179.642,5.681,149.112
C02600=1119.249,-38.447,-49.041,179.642,5.686,149.113
C02601=1119.244,-38.198,-49.053,179.644,5.691,149.113
C02602=1119.239,-37.949,-49.065,179.644,5.696,149.114
C02603=1119.233,-37.699,-49.076,179.644,5.700,149.115
C02604=1119.228,-37.449,-49.088,179.646,5.705,149.116
C02605=1119.222,-37.200,-49.101,179.646,5.710,149.117
C02606=1119.217,-36.950,-49.112,179.647,5.715,149.117
C02607=1119.212,-36.701,-49.124,179.648,5.719,149.118
C02608=1119.207,-36.451,-49.136,179.649,5.725,149.119
C02609=1119.202,-36.201,-49.148,179.650,5.729,149.120
C02610=1119.196,-35.951,-49.160,179.650,5.734,149.121
C02611=1119.191,-35.702,-49.173,179.651,5.739,149.122
C02612=1119.187,-35.452,-49.184,179.652,5.743,149.122
C02613=1119.181,-35.202,-49.196,179.652,5.748,149.123
C02614=1119.176,-34.953,-49.208,179.653,5.753,149.124
C02615=1119.171,-34.703,-49.220,179.653,5.757,149.125
C02616=1119.165,-34.454,-49.233,179.654,5.762,149.126
C02617=1119.161,-34.239,-49.243,179.654,5.766,149.127
C02618=1119.157,-34.023,-49.254,179.654,5.769,149.127
C02619=1119.152,-33.808,-49.264,179.655,5.773,149.128
C02620=1119.148,-33.593,-49.274,179.655,5.777,149.129
C02621=1119.143,-33.378,-49.285,179.655,5.781,149.130
C02622=1119.139,-33.163,-49.295,179.656,5.785,149.130
C02623=1119.134,-32.948,-49.306,179.656,5.788,149.131
C02624=1119.130,-32.733,-49.316,179.656,5.792,149.132
C02625=1119.125,-32.483,-49.328,179.656,5.797,149.133
C02626=1119.119,-32.234,-49.341,179.657,5.802,149.134
C02627=1119.114,-31.984,-49.353,179.657,5.805,149.134
C02628=1119.109,-31.735,-49.365,179.657,5.810,149.135
C02629=1119.103,-31.485,-49.377,179.657,5.814,149.136
C02630=1119.098,-31.235,-49.390,179.657,5.819,149.137
C02631=1119.093,-30.986,-49.402,179.657,5.823,149.138
C02632=1119.089,-30.736,-49.414,179.657,5.827,149.139
C02633=1119.084,-30.486,-49.426,179.658,5.831,149.140
C02634=1119.079,-30.237,-49.438,179.657,5.835,149.141
C02635=1119.073,-29.987,-49.450,179.657,5.840,149.142
C02636=1119.068,-29.737,-49.463,179.657,5.844,149.143
C02637=1119.063,-29.487,-49.475,179.657,5.848,149.144
C02638=1119.057,-29.238,-49.487,179.656,5.853,149.145
C02639=1119.052,-28.989,-49.500,179.656,5.857,149.146
C02640=1119.047,-28.739,-49.512,179.656,5.861,149.147
C02641=1119.042,-28.489,-49.524,179.656,5.865,149.148
C02642=1119.036,-28.240,-49.536,179.655,5.869,149.149
C02643=1119.032,-27.990,-49.549,179.655,5.873,149.150
C02644=1119.027,-27.740,-49.562,179.655,5.878,149.151
C02645=1119.021,-27.490,-49.574,179.655,5.882,149.152
C02646=1119.016,-27.241,-49.586,179.653,5.886,149.153
C02647=1119.011,-26.991,-49.598,179.653,5.890,149.154
C02648=1119.006,-26.742,-49.611,179.653,5.894,149.155
C02649=1119.000,-26.492,-49.624,179.652,5.898,149.156
C02650=1118.995,-26.242,-49.635,179.651,5.903,149.157
C02651=1118.991,-25.992,-49.648,179.651,5.907,149.158
C02652=1118.985,-25.743,-49.661,179.651,5.911,149.159
C02653=1118.980,-25.493,-49.673,179.652,5.917,149.160
C02654=1118.975,-25.244,-49.685,179.652,5.921,149.161
C02655=1118.970,-24.995,-49.698,179.653,5.926,149.162
C02656=1118.964,-24.745,-49.710,179.653,5.931,149.163
C02657=1118.959,-24.495,-49.723,179.654,5.935,149.164
C02658=1118.955,-24.245,-49.736,179.655,5.941,149.165
C02659=1118.949,-23.995,-49.747,179.655,5.946,149.166
C02660=1118.943,-23.746,-49.761,179.656,5.950,149.167
C02661=1118.938,-23.496,-49.773,179.656,5.955,149.167
C02662=1118.933,-23.246,-49.785,179.657,5.960,149.168
C02663=1118.928,-22.997,-49.798,179.658,5.964,149.169
C02664=1118.923,-22.747,-49.811,179.659,5.970,149.170
C02665=1118.918,-22.498,-49.823,179.659,5.975,149.171
C02666=1118.913,-22.248,-49.836,179.660,5.979,149.172
C02667=1118.907,-21.999,-49.848,179.660,5.984,149.173
C02668=1118.902,-21.749,-49.861,179.661,5.989,149.173
C02669=1118.897,-21.499,-49.874,179.661,5.994,149.174
C02670=1118.892,-21.250,-49.886,179.662,5.998,149.175
C02671=1118.887,-21.000,-49.899,179.663,6.003,149.176
C02672=1118.881,-20.750,-49.911,179.663,6.007,149.177
C02673=1118.877,-20.535,-49.923,179.664,6.012,149.178
C02674=1118.872,-20.320,-49.934,179.665,6.016,149.178
C02675=1118.868,-20.106,-49.944,179.665,6.020,149.179
C02676=1118.864,-19.890,-49.956,179.665,6.025,149.180
C02677=1118.859,-19.675,-49.966,179.666,6.028,149.181
C02678=1118.855,-19.461,-49.977,179.667,6.033,149.181
C02679=1118.850,-19.245,-49.988,179.667,6.036,149.182
C02680=1118.846,-19.030,-49.999,179.668,6.041,149.183
C02681=1118.840,-18.781,-50.012,179.668,6.046,149.184
C02682=1118.836,-18.531,-50.025,179.669,6.050,149.184
C02683=1118.831,-18.282,-50.037,179.669,6.055,149.185
C02684=1118.825,-18.032,-50.051,179.670,6.059,149.186
C02685=1118.820,-17.782,-50.064,179.670,6.064,149.187
C02686=1118.815,-17.533,-50.076,179.671,6.068,149.188
C02687=1118.810,-17.284,-50.089,179.672,6.073,149.189
C02688=1118.804,-17.034,-50.102,179.672,6.078,149.190
C02689=1118.800,-16.784,-50.115,179.673,6.083,149.190
C02690=1118.795,-16.535,-50.128,179.673,6.087,149.191
C02691=1118.790,-16.285,-50.140,179.674,6.092,149.192
C02692=1118.784,-16.035,-50.154,179.675,6.096,149.193
C02693=1118.779,-15.786,-50.166,179.675,6.101,149.194
C02694=1118.774,-15.536,-50.179,179.676,6.106,149.195
C02695=1118.769,-15.286,-50.192,179.677,6.110,149.195
C02696=1118.764,-15.037,-50.205,179.677,6.115,149.196
C02697=1118.759,-14.787,-50.218,179.678,6.120,149.197
C02698=1118.753,-14.537,-50.231,179.678,6.124,149.198
C02699=1118.748,-14.288,-50.244,179.679,6.129,149.199
C02700=1118.743,-14.038,-50.256,179.680,6.134,149.200
C02701=1118.738,-13.788,-50.270,179.680,6.138,149.200
C02702=1118.733,-13.539,-50.283,179.681,6.143,149.201
C02703=1118.728,-13.290,-50.296,179.682,6.147,149.202
C02704=1118.723,-13.040,-50.309,179.682,6.152,149.203
C02705=1118.717,-12.790,-50.322,179.683,6.157,149.204
C02706=1118.712,-12.540,-50.336,179.684,6.161,149.205
C02707=1118.707,-12.291,-50.348,179.684,6.166,149.205
C02708=1118.702,-12.042,-50.362,179.685,6.171,149.206
C02709=1118.697,-11.792,-50.375,179.685,6.175,149.207
C02710=1118.692,-11.542,-50.388,179.686,6.180,149.208
C02711=1118.687,-11.292,-50.401,179.687,6.184,149.209
C02712=1118.681,-11.043,-50.414,179.687,6.189,149.210
C02713=1118.677,-10.794,-50.427,179.688,6.193,149.210
C02714=1118.671,-10.544,-50.441,179.689,6.198,149.211
C02715=1118.666,-10.294,-50.453,179.689,6.203,149.212
C02716=1118.661,-10.044,-50.467,179.690,6.207,149.213
C02717=1118.656,-9.795,-50.480,179.691,6.212,149.214
C02718=1118.651,-9.545,-50.494,179.691,6.217,149.215
C02719=1118.646,-9.296,-50.506,179.692,6.221,149.215
C02720=1118.640,-9.046,-50.520,179.693,6.226,149.216
C02721=1118.636,-8.797,-50.533,179.693,6.230,149.217
C02722=1118.630,-8.547,-50.546,179.694,6.235,149.218
C02723=1118.625,-8.297,-50.559,179.694,6.239,149.219
C02724=1118.620,-8.048,-50.573,179.695,6.243,149.219
C02725=1118.615,-7.798,-50.586,179.695,6.248,149.220
C02726=1118.609,-7.548,-50.600,179.696,6.253,149.221
C02727=1118.605,-7.299,-50.613,179.697,6.257,149.222
C02728=1118.599,-7.049,-50.626,179.697,6.262,149.223
C02729=1118.595,-6.834,-50.638,179.698,6.266,149.223
C02730=1118.590,-6.620,-50.649,179.699,6.270,149.224
C02731=1118.586,-6.404,-50.661,179.699,6.273,149.225
C02732=1118.581,-6.190,-50.672,179.699,6.278,149.226
C02733=1118.577,-5.974,-50.684,179.700,6.282,149.226
C02734=1118.573,-5.761,-50.696,179.700,6.285,149.227
C02735=1118.569,-5.545,-50.708,179.701,6.290,149.228
C02736=1118.564,-5.331,-50.719,179.702,6.293,149.228
C02737=1118.559,-5.081,-50.732,179.702,6.298,149.229
C02738=1118.554,-4.832,-50.746,179.703,6.303,149.230
C02739=1118.549,-4.582,-50.759,179.704,6.307,149.231
C02740=1118.544,-4.332,-50.773,179.704,6.312,149.232
C02741=1118.538,-4.082,-50.786,179.705,6.316,149.232
C02742=1118.534,-3.833,-50.800,179.705,6.320,149.233
C02743=1118.528,-3.583,-50.813,179.706,6.325,149.234
C02744=1118.523,-3.334,-50.828,179.706,6.329,149.235
C02745=1118.518,-3.084,-50.840,179.707,6.334,149.236
C02746=1118.513,-2.835,-50.854,179.708,6.338,149.236
C02747=1118.508,-2.585,-50.867,179.708,6.343,149.237
C02748=1118.503,-2.336,-50.881,179.709,6.348,149.238
C02749=1118.497,-2.086,-50.895,179.710,6.352,149.239
C02750=1118.492,-1.836,-50.909,179.710,6.357,149.240
C02751=1118.488,-1.586,-50.922,179.710,6.361,149.241
C02752=1118.482,-1.337,-50.936,179.711,6.365,149.242
C02753=1118.477,-1.087,-50.950,179.712,6.370,149.242
C02754=1118.472,-0.838,-50.963,179.712,6.375,149.243
C02755=1118.467,-0.588,-50.977,179.713,6.379,149.244
C02756=1118.462,-0.339,-50.991,179.714,6.384,149.245
C02757=1118.457,-0.089,-51.004,179.714,6.388,149.246
C02758=1118.452,0.160,-51.018,179.715,6.393,149.246
C02759=1118.446,0.410,-51.031,179.715,6.397,149.247
C02760=1118.441,0.660,-51.045,179.716,6.401,149.248
C02761=1118.437,0.909,-51.059,179.716,6.406,149.249
C02762=1118.431,1.159,-51.072,179.717,6.411,149.250
C02763=1118.426,1.408,-51.087,179.717,6.415,149.251
C02764=1118.421,1.658,-51.101,179.718,6.420,149.251
C02765=1118.416,1.907,-51.115,179.719,6.425,149.252
C02766=1118.411,2.157,-51.128,179.719,6.428,149.253
C02767=1118.406,2.406,-51.142,179.719,6.433,149.254
C02768=1118.401,2.656,-51.156,179.720,6.437,149.255
C02769=1118.396,2.906,-51.170,179.721,6.442,149.256
C02770=1118.391,3.155,-51.183,179.721,6.447,149.256
C02771=1118.386,3.405,-51.197,179.722,6.452,149.257
C02772=1118.381,3.654,-51.211,179.722,6.456,149.258
C02773=1118.375,3.903,-51.225,179.723,6.461,149.259
C02774=1118.370,4.154,-51.239,179.723,6.465,149.260
C02775=1118.365,4.403,-51.253,179.724,6.469,149.261
C02776=1118.360,4.652,-51.266,179.724,6.474,149.261
C02777=1118.355,4.902,-51.281,179.725,6.479,149.262
C02778=1118.350,5.151,-51.295,179.726,6.483,149.263
C02779=1118.345,5.401,-51.309,179.727,6.488,149.264
C02780=1118.340,5.651,-51.323,179.727,6.493,149.265
C02781=1118.335,5.901,-51.337,179.727,6.496,149.266
C02782=1118.330,6.150,-51.351,179.728,6.501,149.267
C02783=1118.324,6.399,-51.365,179.728,6.506,149.267
C02784=1118.320,6.649,-51.379,179.729,6.510,149.268
C02785=1118.315,6.864,-51.391,179.729,6.514,149.269
C02786=1118.311,7.079,-51.403,179.730,6.518,149.270
C02787=1118.306,7.293,-51.415,179.730,6.522,149.270
C02788=1118.303,7.508,-51.427,179.730,6.526,149.271
C02789=1118.298,7.723,-51.440,179.731,6.530,149.272
C02790=1118.293,7.938,-51.451,179.732,6.534,149.273
C02791=1118.289,8.152,-51.464,179.732,6.538,149.273
C02792=1118.284,8.368,-51.476,179.733,6.542,149.274
C02793=1118.279,8.617,-51.490,179.733,6.547,149.275
C02794=1118.275,8.866,-51.504,179.734,6.551,149.276
C02795=1118.270,9.116,-51.518,179.734,6.556,149.277
C02796=1118.265,9.366,-51.532,179.735,6.560,149.277
C02797=1118.260,9.615,-51.546,179.736,6.565,149.278
C02798=1118.254,9.864,-51.560,179.737,6.570,149.279
C02799=1118.249,10.114,-51.575,179.737,6.575,149.280
C02800=1118.244,10.364,-51.589,179.738,6.579,149.281
C02801=1118.239,10.613,-51.603,179.739,6.584,149.282
C02802=1118.234,10.863,-51.617,179.739,6.588,149.282
C02803=1118.229,11.112,-51.631,179.740,6.593,149.283
C02804=1118.224,11.362,-51.646,179.741,6.597,149.284
C02805=1118.218,11.612,-51.661,179.741,6.602,149.285
C02806=1118.214,11.861,-51.676,179.742,6.606,149.285
C02807=1118.209,12.111,-51.690,179.743,6.611,149.286
C02808=1118.203,12.360,-51.704,179.743,6.616,149.287
C02809=1118.198,12.609,-51.718,179.745,6.620,149.288
C02810=1118.193,12.859,-51.732,179.745,6.625,149.289
C02811=1118.188,13.109,-51.747,179.746,6.630,149.290
C02812=1118.183,13.359,-51.761,179.747,6.634,149.290
C02813=1118.178,13.608,-51.775,179.747,6.639,149.291
C02814=1118.174,13.857,-51.790,179.748,6.643,149.292
C02815=1118.168,14.106,-51.804,179.749,6.648,149.293
C02816=1118.163,14.356,-51.818,179.749,6.652,149.294
C02817=1118.158,14.606,-51.833,179.750,6.657,149.294
C02818=1118.152,14.856,-51.847,179.751,6.661,149.295
C02819=1118.148,15.105,-51.862,179.751,6.665,149.296
C02820=1118.143,15.355,-51.877,179.752,6.670,149.297
C02821=1118.138,15.604,-51.891,179.753,6.674,149.297
C02822=1118.133,15.854,-51.905,179.754,6.679,149.298
C02823=1118.128,16.102,-51.920,179.755,6.683,149.299
C02824=1118.123,16.352,-51.934,179.755,6.688,149.300
C02825=1118.117,16.602,-51.949,179.756,6.692,149.301
C02826=1118.112,16.852,-51.963,179.757,6.697,149.301
C02827=1118.107,17.101,-51.978,179.758,6.701,149.302
C02828=1118.102,17.351,-51.993,179.758,6.706,149.303
C02829=1118.097,17.600,-52.007,179.759,6.710,149.303
C02830=1118.092,17.850,-52.022,179.760,6.715,149.304
C02831=1118.087,18.099,-52.037,179.761,6.719,149.305
C02832=1118.082,18.349,-52.051,179.762,6.724,149.306
C02833=1118.078,18.598,-52.066,179.763,6.728,149.307
C02834=1118.072,18.848,-52.081,179.763,6.733,149.307
C02835=1118.067,19.098,-52.095,179.764,6.737,149.308
C02836=1118.062,19.346,-52.110,179.765,6.741,149.309
C02837=1118.057,19.596,-52.124,179.766,6.746,149.310
C02838=1118.051,19.846,-52.140,179.767,6.751,149.310
C02839=1118.046,20.095,-52.154,179.767,6.755,149.311
C02840=1118.042,20.344,-52.169,179.768,6.760,149.312
C02841=1118.037,20.559,-52.182,179.769,6.763,149.312
C02842=1118.033,20.774,-52.194,179.769,6.767,149.313
C02843=1118.029,20.989,-52.207,179.770,6.771,149.314
C02844=1118.025,21.204,-52.220,179.771,6.774,149.314
C02845=1118.020,21.418,-52.233,179.772,6.779,149.315
C02846=1118.016,21.633,-52.245,179.773,6.782,149.316
C02847=1118.012,21.848,-52.258,179.773,6.785,149.316
C02848=1118.007,22.062,-52.271,179.774,6.790,149.317
C02849=1118.002,22.312,-52.285,179.775,6.794,149.317
C02850=1117.997,22.561,-52.300,179.776,6.799,149.318
C02851=1117.992,22.812,-52.315,179.777,6.803,149.319
C02852=1117.987,23.061,-52.330,179.778,6.807,149.320
C02853=1117.982,23.311,-52.344,179.778,6.812,149.321
C02854=1117.977,23.560,-52.360,179.779,6.816,149.321
C02855=1117.972,23.809,-52.375,179.780,6.820,149.322
C02856=1117.967,24.059,-52.389,179.781,6.824,149.322
C02857=1117.962,24.308,-52.405,179.782,6.829,149.323
C02858=1117.957,24.558,-52.419,179.783,6.833,149.324
C02859=1117.951,24.807,-52.435,179.784,6.838,149.325
C02860=1117.947,25.056,-52.450,179.785,6.842,149.325
C02861=1117.942,25.306,-52.464,179.785,6.847,149.326
C02862=1117.936,25.556,-52.480,179.786,6.851,149.327
C02863=1117.932,25.805,-52.494,179.787,6.855,149.328
C02864=1117.926,26.055,-52.509,179.788,6.860,149.328
C02865=1117.922,26.304,-52.524,179.789,6.864,149.329
C02866=1117.916,26.554,-52.539,179.790,6.869,149.330
C02867=1117.911,26.803,-52.554,179.791,6.872,149.330
C02868=1117.906,27.053,-52.570,179.792,6.876,149.331
C02869=1117.902,27.302,-52.585,179.793,6.881,149.332
C02870=1117.896,27.552,-52.600,179.794,6.885,149.332
C02871=1117.891,27.801,-52.615,179.795,6.889,149.333
C02872=1117.886,28.051,-52.631,179.795,6.894,149.334
C02873=1117.881,28.300,-52.645,179.796,6.898,149.334
C02874=1117.876,28.550,-52.661,179.797,6.903,149.335
C02875=1117.871,28.799,-52.676,179.798,6.907,149.336
C02876=1117.866,29.049,-52.692,179.800,6.911,149.336
C02877=1117.862,29.298,-52.707,179.801,6.916,149.337
C02878=1117.856,29.548,-52.721,179.802,6.920,149.338
C02879=1117.851,29.797,-52.736,179.802,6.923,149.338
C02880=1117.846,30.046,-52.752,179.803,6.928,149.339
C02881=1117.841,30.296,-52.767,179.804,6.932,149.340
C02882=1117.836,30.545,-52.783,179.805,6.937,149.341
C02883=1117.831,30.795,-52.797,179.806,6.941,149.341
C02884=1117.826,31.045,-52.813,179.807,6.945,149.342
C02885=1117.821,31.294,-52.828,179.808,6.950,149.343
C02886=1117.816,31.543,-52.843,179.809,6.954,149.343
C02887=1117.811,31.793,-52.859,179.810,6.958,149.344
C02888=1117.807,32.042,-52.874,179.811,6.963,149.344
C02889=1117.801,32.292,-52.890,179.812,6.966,149.345
C02890=1117.796,32.541,-52.906,179.813,6.970,149.346
C02891=1117.791,32.790,-52.921,179.814,6.975,149.346
C02892=1117.786,33.040,-52.936,179.815,6.979,149.347
C02893=1117.781,33.290,-52.951,179.816,6.983,149.348
C02894=1117.776,33.540,-52.966,179.817,6.988,149.348
C02895=1117.771,33.789,-52.982,179.818,6.992,149.349
C02896=1117.766,34.038,-52.997,179.819,6.996,149.350
C02897=1117.762,34.252,-53.011,179.820,6.999,149.350
C02898=1117.757,34.467,-53.024,179.820,7.003,149.351
C02899=1117.753,34.682,-53.037,179.821,7.007,149.351
C02900=1117.749,34.896,-53.051,179.822,7.010,149.352
C02901=1117.745,35.112,-53.064,179.823,7.015,149.353
C02902=1117.740,35.326,-53.078,179.824,7.018,149.353
C02903=1117.736,35.541,-53.091,179.825,7.021,149.354
C02904=1117.732,35.755,-53.104,179.826,7.025,149.354
C02905=1117.727,36.004,-53.120,179.827,7.029,149.355
C02906=1117.721,36.254,-53.135,179.828,7.033,149.355
C02907=1117.717,36.504,-53.151,179.829,7.037,149.356
C02908=1117.712,36.753,-53.166,179.830,7.042,149.357
C02909=1117.706,37.002,-53.182,179.831,7.046,149.357
C02910=1117.701,37.252,-53.197,179.832,7.050,149.358
C02911=1117.696,37.502,-53.213,179.833,7.055,149.359
C02912=1117.692,37.750,-53.229,179.835,7.059,149.359
C02913=1117.687,38.000,-53.245,179.836,7.063,149.360
C02914=1117.682,38.250,-53.261,179.836,7.066,149.360
C02915=1117.676,38.499,-53.276,179.837,7.071,149.361
C02916=1117.671,38.749,-53.292,179.838,7.075,149.362
C02917=1117.667,38.998,-53.307,179.839,7.079,149.362
C02918=1117.662,39.248,-53.323,179.841,7.084,149.363
C02919=1117.656,39.497,-53.339,179.842,7.088,149.363
C02920=1117.652,39.747,-53.355,179.843,7.092,149.364
C02921=1117.646,39.996,-53.371,179.844,7.096,149.365
C02922=1117.641,40.246,-53.386,179.845,7.101,149.365
C02923=1117.637,40.495,-53.402,179.846,7.104,149.366
C02924=1117.632,40.744,-53.418,179.847,7.108,149.366
C02925=1117.626,40.994,-53.434,179.848,7.112,149.367
C02926=1117.622,41.244,-53.449,179.849,7.117,149.368
C02927=1117.617,41.492,-53.466,179.851,7.121,149.368
C02928=1117.611,41.742,-53.481,179.852,7.125,149.369
C02929=1117.606,41.992,-53.497,179.853,7.129,149.369
C02930=1117.602,42.240,-53.513,179.854,7.133,149.370
C02931=1117.597,42.490,-53.529,179.855,7.137,149.371
C02932=1117.592,42.740,-53.545,179.856,7.141,149.371
C02933=1117.587,42.989,-53.561,179.857,7.145,149.372
C02934=1117.582,43.239,-53.577,179.858,7.149,149.372
C02935=1117.577,43.488,-53.592,179.859,7.154,149.373
C02936=1117.572,43.738,-53.609,179.861,7.158,149.374
C02937=1117.567,43.987,-53.625,179.862,7.162,149.374
C02938=1117.561,44.236,-53.640,179.863,7.166,149.375
C02939=1117.557,44.486,-53.657,179.864,7.171,149.376
C02940=1117.551,44.735,-53.672,179.865,7.174,149.376
C02941=1117.547,44.985,-53.689,179.866,7.178,149.377
C02942=1117.542,45.234,-53.705,179.867,7.182,149.377
C02943=1117.537,45.484,-53.721,179.868,7.187,149.378
C02944=1117.532,45.733,-53.737,179.870,7.191,149.378
C02945=1117.527,45.982,-53.753,179.871,7.195,149.379
C02946=1117.522,46.232,-53.769,179.872,7.199,149.380
C02947=1117.517,46.481,-53.785,179.874,7.203,149.380
C02948=1117.512,46.731,-53.802,179.874,7.207,149.381
C02949=1117.507,46.980,-53.817,179.875,7.211,149.381
C02950=1117.502,47.230,-53.834,179.877,7.215,149.382
C02951=1117.497,47.479,-53.850,179.878,7.219,149.382
C02952=1117.492,47.729,-53.866,179.879,7.223,149.383
C02953=1117.488,47.943,-53.880,179.880,7.227,149.384
C02954=1117.484,48.157,-53.893,179.881,7.230,149.384
C02955=1117.480,48.372,-53.908,179.882,7.234,149.385
C02956=1117.475,48.587,-53.922,179.883,7.237,149.385
C02957=1117.471,48.801,-53.936,179.884,7.241,149.385
C02958=1117.466,49.016,-53.949,179.885,7.244,149.386
C02959=1117.463,49.230,-53.964,179.886,7.248,149.387
C02960=1117.459,49.444,-53.978,179.887,7.252,149.387
C02961=1117.453,49.694,-53.993,179.888,7.255,149.387
C02962=1117.448,49.944,-54.011,179.889,7.259,149.388
C02963=1117.444,50.193,-54.027,179.890,7.263,149.389
C02964=1117.438,50.442,-54.043,179.892,7.267,149.389
C02965=1117.434,50.692,-54.060,179.893,7.272,149.390
C02966=1117.429,50.941,-54.076,179.895,7.275,149.390
C02967=1117.424,51.191,-54.092,179.896,7.280,149.391
C02968=1117.419,51.440,-54.108,179.897,7.284,149.392
C02969=1117.414,51.689,-54.125,179.898,7.288,149.392
C02970=1117.408,51.939,-54.141,179.899,7.291,149.393
C02971=1117.404,52.188,-54.158,179.900,7.295,149.393
C02972=1117.399,52.438,-54.174,179.901,7.300,149.394
C02973=1117.394,52.687,-54.191,179.903,7.304,149.394
C02974=1117.389,52.937,-54.207,179.904,7.308,149.395
C02975=1117.384,53.186,-54.223,179.905,7.312,149.395
C02976=1117.379,53.435,-54.240,179.907,7.316,149.396
C02977=1117.375,53.685,-54.257,179.908,7.320,149.396
C02978=1117.369,53.934,-54.272,179.909,7.323,149.397
C02979=1117.364,54.184,-54.290,179.910,7.328,149.398
C02980=1117.359,54.433,-54.306,179.911,7.332,149.398
C02981=1117.354,54.682,-54.323,179.912,7.336,149.399
C02982=1117.350,54.932,-54.339,179.914,7.340,149.399
C02983=1117.344,55.181,-54.356,179.915,7.344,149.400
C02984=1117.339,55.431,-54.372,179.917,7.348,149.400
C02985=1117.334,55.680,-54.388,179.918,7.352,149.401
C02986=1117.329,55.929,-54.406,179.919,7.356,149.401
C02987=1117.325,56.179,-54.422,179.920,7.360,149.402
C02988=1117.319,56.428,-54.439,179.921,7.364,149.402
C02989=1117.315,56.677,-54.455,179.922,7.368,149.403
C02990=1117.310,56.927,-54.473,179.924,7.372,149.403
C02991=1117.305,57.176,-54.489,179.925,7.376,149.404
C02992=1117.300,57.425,-54.506,179.927,7.380,149.404
C02993=1117.295,57.675,-54.523,179.928,7.384,149.405
C02994=1117.290,57.924,-54.539,179.929,7.388,149.406
C02995=1117.285,58.173,-54.556,179.930,7.392,149.406
C02996=1117.280,58.423,-54.573,179.931,7.396,149.407
C02997=1117.276,58.673,-54.590,179.932,7.400,149.407
C02998=1117.270,58.922,-54.607,179.934,7.404,149.408
C02999=1117.265,59.171,-54.623,179.936,7.408,149.408
C03000=1117.261,59.421,-54.640,179.937,7.412,149.409
C03001=1117.255,59.670,-54.657,179.938,7.416,149.409
C03002=1117.251,59.919,-54.674,179.939,7.420,149.410
C03003=1117.245,60.169,-54.691,179.941,7.424,149.410
C03004=1117.241,60.419,-54.707,179.941,7.428,149.411
C03005=1117.236,60.667,-54.724,179.943,7.432,149.411
C03006=1117.231,60.917,-54.741,179.945,7.436,149.412
C03007=1117.226,61.167,-54.758,179.946,7.440,149.412
C03008=1117.221,61.416,-54.775,179.947,7.444,149.413
C03009=1117.217,61.630,-54.789,179.948,7.447,149.413
C03010=1117.212,61.845,-54.804,179.950,7.451,149.414
C03011=1117.209,62.059,-54.818,179.951,7.454,149.414
C03012=1117.204,62.273,-54.834,179.951,7.457,149.415
C03013=1117.200,62.488,-54.848,179.953,7.461,149.415
C03014=1117.195,62.702,-54.863,179.954,7.465,149.416
C03015=1117.192,62.917,-54.877,179.955,7.468,149.416
C03016=1117.187,63.131,-54.892,179.956,7.472,149.417
C03017=1117.183,63.381,-54.908,179.958,7.475,149.417
C03018=1117.177,63.631,-54.926,179.959,7.480,149.418
C03019=1117.173,63.879,-54.943,179.960,7.484,149.418
C03020=1117.167,64.129,-54.960,179.961,7.487,149.418
C03021=1117.163,64.378,-54.977,179.962,7.491,149.419
C03022=1117.158,64.628,-54.994,179.964,7.495,149.420
C03023=1117.153,64.877,-55.011,179.966,7.499,149.420
C03024=1117.148,65.126,-55.028,179.967,7.503,149.421
C03025=1117.142,65.376,-55.045,179.968,7.507,149.421
C03026=1117.138,65.624,-55.063,179.969,7.511,149.422
C03027=1117.133,65.874,-55.080,179.971,7.515,149.422
C03028=1117.129,66.124,-55.097,179.972,7.519,149.423
C03029=1117.124,66.373,-55.115,179.974,7.523,149.423
C03030=1117.119,66.622,-55.131,179.975,7.527,149.424
C03031=1117.114,66.872,-55.149,179.976,7.530,149.424
C03032=1117.108,67.121,-55.166,179.977,7.535,149.425
C03033=1117.104,67.370,-55.183,179.979,7.539,149.425
C03034=1117.099,67.620,-55.200,179.980,7.543,149.426
C03035=1117.094,67.869,-55.218,179.981,7.547,149.426
C03036=1117.089,68.119,-55.235,179.983,7.551,149.427
C03037=1117.084,68.368,-55.253,179.985,7.555,149.427
C03038=1117.079,68.618,-55.270,179.986,7.559,149.428
C03039=1117.075,68.867,-55.287,179.987,7.563,149.428
C03040=1117.070,69.116,-55.305,179.989,7.567,149.429
C03041=1117.064,69.365,-55.322,179.989,7.570,149.429
C03042=1117.060,69.614,-55.339,179.991,7.574,149.430
C03043=1117.055,69.864,-55.356,179.992,7.578,149.430
C03044=1117.050,70.113,-55.374,179.994,7.582,149.431
C03045=1117.045,70.363,-55.391,179.995,7.586,149.431
C03046=1117.040,70.612,-55.409,179.997,7.590,149.432
C03047=1117.035,70.862,-55.426,179.998,7.594,149.432
C03048=1117.030,71.111,-55.444,179.999,7.598,149.433
C03049=1117.026,71.360,-55.461,-179.999,7.602,149.433
C03050=1117.021,71.609,-55.479,-179.997,7.606,149.434
C03051=1117.016,71.859,-55.497,-179.996,7.610,149.434
C03052=1117.011,72.108,-55.514,-179.995,7.614,149.435
C03053=1117.006,72.357,-55.531,-179.993,7.618,149.435
C03054=1117.001,72.607,-55.549,-179.992,7.621,149.436
C03055=1116.996,72.856,-55.567,-179.991,7.626,149.436
C03056=1116.991,73.105,-55.585,-179.990,7.630,149.437
C03057=1116.987,73.355,-55.601,-179.988,7.633,149.437
C03058=1116.982,73.604,-55.619,-179.987,7.638,149.438
C03059=1116.977,73.854,-55.637,-179.985,7.642,149.438
C03060=1116.972,74.103,-55.655,-179.984,7.646,149.439
C03061=1116.967,74.352,-55.673,-179.982,7.649,149.439
C03062=1116.962,74.601,-55.690,-179.981,7.654,149.440
C03063=1116.958,74.851,-55.707,-179.979,7.658,149.440
C03064=1116.953,75.100,-55.725,-179.978,7.662,149.440
C03065=1116.945,75.459,-55.751,-179.976,7.667,149.441
C03066=1116.938,75.818,-55.777,-179.974,7.673,149.442
C03067=1116.931,76.176,-55.802,-179.972,7.679,149.443
C03068=1116.924,76.535,-55.828,-179.969,7.685,149.443
C03069=1116.919,76.815,-55.847,-179.968,7.689,149.444
C03070=1116.914,77.064,-55.865,-179.967,7.692,149.444
C03071=1116.909,77.313,-55.883,-179.966,7.696,149.445
C03072=1116.904,77.563,-55.900,-179.965,7.699,149.445
C03073=1116.899,77.812,-55.918,-179.964,7.704,149.446
C03074=1116.894,78.061,-55.936,-179.964,7.707,149.447
C03075=1116.889,78.310,-55.954,-179.962,7.711,149.447
C03076=1116.884,78.560,-55.972,-179.962,7.715,149.448
C03077=1116.879,78.809,-55.990,-179.960,7.718,149.448
C03078=1116.875,79.059,-56.008,-179.959,7.722,149.449
C03079=1116.870,79.308,-56.026,-179.958,7.726,149.449
C03080=1116.865,79.558,-56.044,-179.957,7.729,149.450
C03081=1116.861,79.807,-56.061,-179.956,7.733,149.450
C03082=1116.856,80.056,-56.079,-179.955,7.737,149.451
C03083=1116.851,80.305,-56.097,-179.954,7.741,149.451
C03084=1116.846,80.554,-56.115,-179.953,7.744,149.452
C03085=1116.841,80.803,-56.133,-179.952,7.748,149.453
C03086=1116.835,81.053,-56.152,-179.951,7.751,149.453
C03087=1116.831,81.303,-56.170,-179.950,7.756,149.454
C03088=1116.826,81.552,-56.188,-179.949,7.759,149.454
C03089=1116.821,81.801,-56.206,-179.947,7.763,149.455
C03090=1116.816,82.050,-56.224,-179.946,7.767,149.455
C03091=1116.811,82.299,-56.242,-179.945,7.770,149.456
C03092=1116.807,82.548,-56.260,-179.944,7.774,149.456
C03093=1116.802,82.798,-56.278,-179.943,7.778,149.457
C03094=1116.797,83.048,-56.296,-179.942,7.782,149.457
C03095=1116.792,83.297,-56.314,-179.941,7.786,149.458
C03096=1116.787,83.546,-56.332,-179.940,7.789,149.459
C03097=1116.783,83.795,-56.350,-179.938,7.793,149.459
C03098=1116.778,84.044,-56.368,-179.937,7.797,149.460
C03099=1116.773,84.293,-56.386,-179.936,7.801,149.460
C03100=1116.768,84.543,-56.405,-179.935,7.804,149.461
C03101=1116.763,84.793,-56.423,-179.934,7.809,149.461
C03102=1116.758,85.042,-56.441,-179.933,7.812,149.462
C03103=1116.753,85.291,-56.459,-179.931,7.816,149.462
C03104=1116.748,85.540,-56.477,-179.930,7.820,149.463
C03105=1116.744,85.790,-56.496,-179.929,7.823,149.463
C03106=1116.739,86.039,-56.514,-179.928,7.827,149.464
C03107=1116.734,86.288,-56.532,-179.926,7.831,149.464
C03108=1116.729,86.537,-56.551,-179.925,7.834,149.465
C03109=1116.724,86.787,-56.569,-179.924,7.839,149.465
C03110=1116.719,87.036,-56.587,-179.923,7.843,149.466
C03111=1116.715,87.285,-56.606,-179.921,7.846,149.466
C03112=1116.710,87.534,-56.624,-179.920,7.850,149.467
C03113=1116.705,87.784,-56.642,-179.919,7.854,149.467
C03114=1116.700,88.034,-56.661,-179.917,7.858,149.468
C03115=1116.695,88.283,-56.679,-179.916,7.862,149.468
C03116=1116.690,88.531,-56.697,-179.915,7.865,149.469
C03117=1116.686,88.781,-56.716,-179.914,7.869,149.469
C03118=1116.682,88.995,-56.731,-179.913,7.872,149.470
C03119=1116.677,89.210,-56.747,-179.911,7.876,149.470
C03120=1116.673,89.424,-56.764,-179.910,7.879,149.470
C03121=1116.669,89.638,-56.779,-179.909,7.882,149.471
C03122=1116.665,89.852,-56.795,-179.907,7.886,149.471
C03123=1116.661,90.066,-56.811,-179.906,7.889,149.472
C03124=1116.656,90.281,-56.826,-179.905,7.892,149.472
C03125=1116.652,90.495,-56.843,-179.905,7.895,149.473
C03126=1116.647,90.744,-56.861,-179.903,7.899,149.473
C03127=1116.643,90.993,-56.880,-179.901,7.903,149.473
C03128=1116.638,91.243,-56.898,-179.900,7.907,149.474
C03129=1116.632,91.492,-56.916,-179.898,7.911,149.474
C03130=1116.628,91.741,-56.935,-179.897,7.915,149.475
C03131=1116.623,91.991,-56.953,-179.895,7.919,149.475
C03132=1116.618,92.239,-56.973,-179.894,7.922,149.476
C03133=1116.614,92.489,-56.991,-179.893,7.926,149.476
C03134=1116.609,92.738,-57.009,-179.891,7.930,149.477
C03135=1116.604,92.987,-57.028,-179.890,7.934,149.477
C03136=1116.599,93.237,-57.047,-179.888,7.938,149.478
C03137=1116.595,93.486,-57.065,-179.886,7.942,149.478
C03138=1116.589,93.735,-57.084,-179.885,7.946,149.478
C03139=1116.585,93.985,-57.103,-179.883,7.950,149.479
C03140=1116.579,94.234,-57.122,-179.882,7.954,149.479
C03141=1116.575,94.483,-57.141,-179.881,7.957,149.480
C03142=1116.570,94.732,-57.159,-179.880,7.961,149.480
C03143=1116.565,94.981,-57.178,-179.878,7.965,149.481
C03144=1116.561,95.231,-57.196,-179.876,7.969,149.481
C03145=1116.555,95.480,-57.216,-179.875,7.972,149.482
C03146=1116.550,95.729,-57.234,-179.873,7.976,149.482
C03147=1116.546,95.979,-57.253,-179.872,7.980,149.483
C03148=1116.541,96.228,-57.271,-179.870,7.984,149.483
C03149=1116.537,96.477,-57.290,-179.868,7.988,149.483
C03150=1116.531,96.726,-57.310,-179.866,7.992,149.484
C03151=1116.527,96.976,-57.328,-179.865,7.995,149.484
C03152=1116.522,97.225,-57.347,-179.863,7.999,149.484
C03153=1116.517,97.473,-57.366,-179.861,8.003,149.485
C03154=1116.512,97.724,-57.385,-179.860,8.007,149.485
C03155=1116.508,97.972,-57.403,-179.858,8.011,149.486
C03156=1116.503,98.222,-57.423,-179.857,8.015,149.486
C03157=1116.498,98.471,-57.441,-179.855,8.019,149.487
C03158=1116.493,98.720,-57.461,-179.853,8.022,149.487
C03159=1116.489,98.969,-57.479,-179.851,8.026,149.487
C03160=1116.484,99.219,-57.498,-179.850,8.030,149.488
C03161=1116.478,99.468,-57.518,-179.848,8.034,149.488
C03162=1116.474,99.717,-57.537,-179.847,8.038,149.489
C03163=1116.469,99.966,-57.556,-179.845,8.041,149.489
C03164=1116.465,100.216,-57.574,-179.843,8.045,149.489
C03165=1116.459,100.465,-57.594,-179.841,8.049,149.490
C03166=1116.455,100.714,-57.613,-179.840,8.053,149.490
C03167=1116.450,100.963,-57.632,-179.837,8.057,149.490
C03168=1116.445,101.213,-57.651,-179.835,8.061,149.491
C03169=1116.440,101.462,-57.670,-179.834,8.065,149.491
C03170=1116.435,101.711,-57.689,-179.832,8.069,149.491
C03171=1116.430,101.960,-57.709,-179.830,8.072,149.492
C03172=1116.426,102.209,-57.728,-179.829,8.076,149.492
C03173=1116.421,102.458,-57.747,-179.827,8.080,149.492
C03174=1116.417,102.672,-57.763,-179.825,8.084,149.493
C03175=1116.412,102.887,-57.780,-179.823,8.086,149.493
C03176=1116.409,103.101,-57.796,-179.821,8.090,149.493
C03177=1116.404,103.315,-57.813,-179.820,8.093,149.494
C03178=1116.400,103.529,-57.829,-179.818,8.097,149.494
C03179=1116.396,103.743,-57.846,-179.817,8.100,149.494
C03180=1116.392,103.957,-57.862,-179.815,8.103,149.495
C03181=1116.388,104.172,-57.879,-179.814,8.106,149.495
C03182=1116.383,104.421,-57.899,-179.812,8.111,149.495
C03183=1116.379,104.671,-57.918,-179.810,8.114,149.496
C03184=1116.373,104.919,-57.937,-179.808,8.118,149.496
C03185=1116.369,105.169,-57.957,-179.806,8.121,149.496
C03186=1116.363,105.418,-57.976,-179.804,8.125,149.497
C03187=1116.359,105.667,-57.995,-179.802,8.129,149.497
C03188=1116.355,105.917,-58.015,-179.800,8.132,149.497
C03189=1116.349,106.166,-58.034,-179.798,8.137,149.498
C03190=1116.345,106.415,-58.054,-179.796,8.140,149.498
C03191=1116.341,106.664,-58.073,-179.794,8.144,149.498
C03192=1116.335,106.913,-58.093,-179.792,8.148,149.498
C03193=1116.331,107.162,-58.112,-179.790,8.151,149.499
C03194=1116.325,107.411,-58.132,-179.788,8.156,149.499
C03195=1116.321,107.661,-58.151,-179.786,8.160,149.499
C03196=1116.317,107.910,-58.170,-179.784,8.163,149.500
C03197=1116.311,108.159,-58.190,-179.782,8.167,149.500
C03198=1116.307,108.408,-58.209,-179.780,8.170,149.500
C03199=1116.302,108.657,-58.230,-179.778,8.175,149.500
C03200=1116.297,108.906,-58.249,-179.775,8.178,149.501
C03201=1116.292,109.156,-58.269,-179.773,8.182,149.501
C03202=1116.287,109.405,-58.288,-179.771,8.185,149.501
C03203=1116.283,109.655,-58.307,-179.770,8.189,149.501
C03204=1116.278,109.903,-58.327,-179.767,8.193,149.502
C03205=1116.273,110.152,-58.347,-179.765,8.197,149.502
C03206=1116.269,110.402,-58.367,-179.763,8.200,149.502
C03207=1116.263,110.651,-58.386,-179.761,8.204,149.502
C03208=1116.259,110.900,-58.406,-179.758,8.208,149.503
C03209=1116.254,111.149,-58.426,-179.756,8.212,149.503
C03210=1116.249,111.399,-58.446,-179.755,8.216,149.503
C03211=1116.244,111.647,-58.466,-179.753,8.218,149.504
C03212=1116.240,111.897,-58.485,-179.751,8.222,149.504
C03213=1116.235,112.146,-58.505,-179.749,8.226,149.504
C03214=1116.231,112.395,-58.525,-179.747,8.229,149.504
C03215=1116.225,112.644,-58.544,-179.745,8.233,149.505
C03216=1116.221,112.893,-58.565,-179.744,8.236,149.505
C03217=1116.216,113.143,-58.585,-179.742,8.239,149.505
C03218=1116.211,113.392,-58.604,-179.740,8.243,149.505
C03219=1116.206,113.640,-58.624,-179.738,8.246,149.506
C03220=1116.201,113.890,-58.644,-179.737,8.250,149.506
C03221=1116.197,114.139,-58.664,-179.735,8.253,149.506
C03222=1116.192,114.389,-58.684,-179.733,8.256,149.507
C03223=1116.188,114.637,-58.704,-179.731,8.260,149.507
C03224=1116.183,114.886,-58.724,-179.729,8.264,149.507
C03225=1116.178,115.135,-58.744,-179.727,8.267,149.507
C03226=1116.173,115.385,-58.764,-179.726,8.270,149.508
C03227=1116.169,115.634,-58.784,-179.724,8.274,149.508
C03228=1116.163,115.884,-58.804,-179.722,8.277,149.508
C03229=1116.158,116.132,-58.824,-179.720,8.281,149.509
C03230=1116.154,116.347,-58.841,-179.719,8.284,149.509
C03231=1116.151,116.561,-58.858,-179.717,8.286,149.509
C03232=1116.147,116.774,-58.875,-179.716,8.289,149.509
C03233=1116.142,116.988,-58.893,-179.714,8.293,149.510
C03234=1116.138,117.203,-58.910,-179.713,8.296,149.510
C03235=1116.134,117.417,-58.927,-179.711,8.298,149.510
C03236=1116.130,117.631,-58.945,-179.710,8.301,149.510
C03237=1116.126,117.845,-58.962,-179.708,8.305,149.511
C03238=1116.121,118.094,-58.982,-179.706,8.307,149.511
C03239=1116.117,118.343,-59.002,-179.704,8.311,149.511
C03240=1116.112,118.592,-59.023,-179.703,8.315,149.511
C03241=1116.107,118.842,-59.042,-179.701,8.318,149.512
C03242=1116.103,119.091,-59.063,-179.699,8.321,149.512
C03243=1116.098,119.340,-59.084,-179.697,8.324,149.512
C03244=1116.093,119.589,-59.103,-179.696,8.328,149.513
C03245=1116.089,119.838,-59.124,-179.693,8.332,149.513
C03246=1116.084,120.087,-59.144,-179.692,8.334,149.513
C03247=1116.078,120.336,-59.165,-179.690,8.338,149.513
C03248=1116.074,120.585,-59.184,-179.688,8.342,149.514
C03249=1116.069,120.834,-59.205,-179.687,8.344,149.514
C03250=1116.065,121.083,-59.225,-179.685,8.348,149.514
C03251=1116.060,121.332,-59.245,-179.683,8.351,149.514
C03252=1116.055,121.582,-59.266,-179.681,8.355,149.515
C03253=1116.050,121.831,-59.286,-179.680,8.358,149.515
C03254=1116.046,122.080,-59.306,-179.678,8.362,149.515
C03255=1116.041,122.329,-59.327,-179.676,8.365,149.515
C03256=1116.036,122.578,-59.348,-179.674,8.369,149.516
C03257=1116.032,122.828,-59.367,-179.673,8.372,149.516
C03258=1116.027,123.077,-59.388,-179.670,8.375,149.516
C03259=1116.022,123.326,-59.409,-179.668,8.379,149.517
C03260=1116.018,123.575,-59.429,-179.667,8.381,149.517
C03261=1116.013,123.824,-59.449,-179.665,8.385,149.517
C03262=1116.008,124.073,-59.470,-179.663,8.389,149.517
C03263=1116.003,124.322,-59.491,-179.662,8.391,149.518
C03264=1115.999,124.571,-59.511,-179.660,8.395,149.518
C03265=1115.994,124.821,-59.531,-179.658,8.398,149.518
C03266=1115.989,125.070,-59.552,-179.656,8.402,149.519
C03267=1115.985,125.319,-59.572,-179.655,8.405,149.519
C03268=1115.979,125.568,-59.593,-179.653,8.409,149.519
C03269=1115.975,125.817,-59.613,-179.650,8.412,149.519
C03270=1115.970,126.066,-59.634,-179.649,8.415,149.520
C03271=1115.965,126.315,-59.655,-179.647,8.419,149.520
C03272=1115.961,126.564,-59.675,-179.645,8.422,149.520
C03273=1115.956,126.814,-59.696,-179.644,8.425,149.520
C03274=1115.951,127.062,-59.717,-179.642,8.429,149.521
C03275=1115.946,127.312,-59.737,-179.640,8.432,149.521
C03276=1115.942,127.561,-59.758,-179.639,8.435,149.521
C03277=1115.937,127.810,-59.779,-179.637,8.438,149.522
C03278=1115.932,128.059,-59.799,-179.635,8.442,149.522
C03279=1115.928,128.307,-59.820,-179.634,8.445,149.522
C03280=1115.923,128.556,-59.841,-179.632,8.449,149.522
C03281=1115.918,128.805,-59.862,-179.630,8.452,149.523
C03282=1115.914,129.055,-59.883,-179.629,8.455,149.523
C03283=1115.909,129.304,-59.903,-179.626,8.459,149.523
C03284=1115.904,129.554,-59.924,-179.624,8.462,149.524
C03285=1115.900,129.803,-59.945,-179.623,8.465,149.524
C03286=1115.895,130.016,-59.963,-179.621,8.468,149.524
C03287=1115.891,130.230,-59.981,-179.620,8.471,149.524
C03288=1115.887,130.444,-59.999,-179.618,8.474,149.525
C03289=1115.883,130.658,-60.016,-179.617,8.477,149.525
C03290=1115.880,130.872,-60.034,-179.616,8.480,149.525
C03291=1115.875,131.086,-60.052,-179.614,8.482,149.525
C03292=1115.871,131.301,-60.070,-179.613,8.485,149.526
C03293=1115.867,131.514,-60.088,-179.611,8.488,149.526
C03294=1115.862,131.763,-60.109,-179.609,8.491,149.526
C03295=1115.858,132.013,-60.130,-179.608,8.495,149.526
C03296=1115.853,132.261,-60.152,-179.606,8.498,149.527
C03297=1115.849,132.510,-60.172,-179.604,8.501,149.527
C03298=1115.844,132.759,-60.193,-179.602,8.505,149.527
C03299=1115.838,133.009,-60.214,-179.601,8.508,149.528
C03300=1115.834,133.257,-60.235,-179.599,8.511,149.528
C03301=1115.829,133.506,-60.256,-179.597,8.515,149.528
C03302=1115.824,133.756,-60.277,-179.596,8.518,149.528
C03303=1115.820,134.005,-60.299,-179.594,8.521,149.529
C03304=1115.815,134.254,-60.320,-179.592,8.525,149.529
C03305=1115.811,134.503,-60.340,-179.591,8.528,149.529
C03306=1115.806,134.751,-60.362,-179.589,8.532,149.530
C03307=1115.801,135.001,-60.383,-179.586,8.535,149.530
C03308=1115.797,135.250,-60.403,-179.585,8.538,149.530
C03309=1115.792,135.499,-60.425,-179.583,8.542,149.530
C03310=1115.787,135.748,-60.446,-179.582,8.544,149.531
C03311=1115.783,135.997,-60.467,-179.580,8.548,149.531
C03312=1115.778,136.247,-60.488,-179.578,8.552,149.531
C03313=1115.773,136.496,-60.509,-179.577,8.554,149.532
C03314=1115.768,136.744,-60.531,-179.575,8.558,149.532
C03315=1115.764,136.993,-60.551,-179.573,8.562,149.532
C03316=1115.759,137.243,-60.573,-179.572,8.564,149.533
C03317=1115.754,137.492,-60.594,-179.570,8.568,149.533
C03318=1115.750,137.740,-60.615,-179.568,8.572,149.533
C03319=1115.745,137.990,-60.636,-179.567,8.575,149.534
C03320=1115.741,138.239,-60.658,-179.565,8.578,149.534
C03321=1115.735,138.488,-60.679,-179.563,8.581,149.534
C03322=1115.731,138.737,-60.701,-179.562,8.585,149.535
C03323=1115.726,138.986,-60.721,-179.560,8.588,149.535
C03324=1115.722,139.235,-60.744,-179.559,8.592,149.535
C03325=1115.717,139.484,-60.765,-179.557,8.595,149.535
C03326=1115.712,139.733,-60.786,-179.555,8.599,149.536
C03327=1115.708,139.982,-60.808,-179.554,8.602,149.536
C03328=1115.703,140.231,-60.829,-179.551,8.605,149.536
C03329=1115.698,140.480,-60.850,-179.550,8.609,149.537
C03330=1115.693,140.729,-60.872,-179.548,8.612,149.537
C03331=1115.689,140.979,-60.893,-179.547,8.616,149.537
C03332=1115.684,141.227,-60.915,-179.545,8.618,149.538
C03333=1115.680,141.476,-60.935,-179.543,8.622,149.538
C03334=1115.675,141.725,-60.957,-179.542,8.626,149.538
C03335=1115.670,141.974,-60.979,-179.540,8.628,149.539
C03336=1115.665,142.223,-61.000,-179.538,8.632,149.539
C03337=1115.661,142.473,-61.022,-179.536,8.636,149.539
C03338=1115.656,142.721,-61.044,-179.535,8.639,149.540
C03339=1115.651,142.970,-61.065,-179.533,8.642,149.540
C03340=1115.647,143.220,-61.086,-179.532,8.645,149.540
C03341=1115.642,143.468,-61.108,-179.530,8.649,149.541
C03342=1115.638,143.682,-61.127,-179.529,8.652,149.541
C03343=1115.634,143.896,-61.145,-179.528,8.655,149.541
C03344=1115.630,144.110,-61.164,-179.526,8.657,149.541
C03345=1115.627,144.324,-61.182,-179.525,8.661,149.542
C03346=1115.622,144.538,-61.201,-179.523,8.664,149.542
C03347=1115.619,144.752,-61.219,-179.522,8.667,149.542
C03348=1115.614,144.965,-61.238,-179.521,8.670,149.543
C03349=1115.610,145.179,-61.257,-179.519,8.672,149.543
C03350=1115.605,145.428,-61.279,-179.517,8.676,149.543
C03351=1115.601,145.677,-61.301,-179.515,8.680,149.543
C03352=1115.596,145.926,-61.321,-179.512,8.684,149.544
C03353=1115.592,146.176,-61.343,-179.510,8.687,149.544
C03354=1115.587,146.424,-61.365,-179.508,8.691,149.544
C03355=1115.583,146.674,-61.387,-179.506,8.695,149.545
C03356=1115.577,146.923,-61.409,-179.504,8.699,149.545
C03357=1115.572,147.171,-61.431,-179.502,8.702,149.545
C03358=1115.568,147.421,-61.453,-179.500,8.706,149.545
C03359=1115.563,147.669,-61.475,-179.498,8.709,149.546
C03360=1115.559,147.918,-61.497,-179.495,8.714,149.546
C03361=1115.554,148.167,-61.518,-179.493,8.717,149.546
C03362=1115.550,148.416,-61.540,-179.491,8.721,149.546
C03363=1115.545,148.665,-61.562,-179.489,8.724,149.546
C03364=1115.541,148.914,-61.584,-179.486,8.727,149.547
C03365=1115.536,149.163,-61.606,-179.484,8.731,149.547
C03366=1115.531,149.412,-61.627,-179.481,8.735,149.547
C03367=1115.527,149.661,-61.649,-179.479,8.738,149.547
C03368=1115.522,149.910,-61.671,-179.477,8.742,149.547
C03369=1115.517,150.159,-61.694,-179.475,8.745,149.548
C03370=1115.512,150.408,-61.715,-179.473,8.749,149.548
C03371=1115.508,150.657,-61.738,-179.471,8.752,149.548
C03372=1115.503,150.906,-61.759,-179.468,8.757,149.548
C03373=1115.499,151.155,-61.781,-179.466,8.760,149.548
C03374=1115.494,151.404,-61.803,-179.464,8.763,149.549
C03375=1115.489,151.654,-61.826,-179.462,8.767,149.549
C03376=1115.485,151.902,-61.848,-179.460,8.770,149.549
C03377=1115.480,152.151,-61.870,-179.457,8.774,149.549
C03378=1115.476,152.400,-61.892,-179.455,8.777,149.549
C03379=1115.471,152.649,-61.914,-179.453,8.780,149.550
C03380=1115.466,152.899,-61.936,-179.451,8.784,149.550
C03381=1115.461,153.147,-61.959,-179.449,8.787,149.550
C03382=1115.457,153.396,-61.981,-179.446,8.790,149.550
C03383=1115.452,153.645,-62.003,-179.444,8.794,149.550
C03384=1115.447,153.894,-62.025,-179.442,8.797,149.551
C03385=1115.443,154.143,-62.048,-179.439,8.802,149.551
C03386=1115.438,154.392,-62.070,-179.437,8.805,149.551
C03387=1115.434,154.641,-62.092,-179.435,8.808,149.551
C03388=1115.428,154.890,-62.114,-179.433,8.812,149.551
C03389=1115.424,155.139,-62.137,-179.430,8.815,149.551
C03390=1115.420,155.388,-62.159,-179.428,8.818,149.552
C03391=1115.415,155.637,-62.181,-179.426,8.822,149.552
C03392=1115.411,155.886,-62.204,-179.423,8.825,149.552
C03393=1115.406,156.134,-62.225,-179.421,8.828,149.552
C03394=1115.401,156.383,-62.249,-179.419,8.831,149.552
C03395=1115.397,156.633,-62.271,-179.417,8.835,149.552
C03396=1115.392,156.881,-62.293,-179.415,8.838,149.553
C03397=1115.387,157.130,-62.316,-179.413,8.841,149.553
C03398=1115.383,157.345,-62.335,-179.411,8.844,149.553
C03399=1115.379,157.558,-62.355,-179.409,8.847,149.553
C03400=1115.375,157.771,-62.373,-179.407,8.850,149.553
C03401=1115.372,157.985,-62.393,-179.405,8.852,149.553
C03402=1115.368,158.199,-62.412,-179.403,8.855,149.553
C03403=1115.364,158.413,-62.432,-179.401,8.858,149.553
C03404=1115.360,158.627,-62.451,-179.399,8.861,149.554
C03405=1115.356,158.840,-62.471,-179.397,8.864,149.554
C03406=1115.351,159.089,-62.492,-179.395,8.867,149.554
C03407=1115.346,159.338,-62.516,-179.393,8.870,149.554
C03408=1115.342,159.587,-62.538,-179.391,8.873,149.554
C03409=1115.337,159.836,-62.561,-179.388,8.876,149.554
C03410=1115.332,160.085,-62.583,-179.386,8.880,149.555
C03411=1115.328,160.334,-62.606,-179.384,8.883,149.555
C03412=1115.324,160.583,-62.628,-179.382,8.887,149.555
C03413=1115.318,160.832,-62.651,-179.379,8.890,149.555
C03414=1115.314,161.080,-62.674,-179.377,8.893,149.555
C03415=1115.309,161.330,-62.696,-179.374,8.896,149.555
C03416=1115.305,161.579,-62.719,-179.373,8.899,149.555
C03417=1115.300,161.827,-62.742,-179.371,8.902,149.555
C03418=1115.296,162.076,-62.764,-179.368,8.905,149.555
C03419=1115.291,162.325,-62.788,-179.366,8.909,149.556
C03420=1115.287,162.574,-62.810,-179.363,8.912,149.556
C03421=1115.281,162.823,-62.833,-179.361,8.915,149.556
C03422=1115.277,163.072,-62.855,-179.359,8.918,149.556
C03423=1115.273,163.321,-62.879,-179.357,8.921,149.556
C03424=1115.269,163.570,-62.902,-179.355,8.924,149.556
C03425=1115.264,163.819,-62.924,-179.352,8.927,149.556
C03426=1115.259,164.068,-62.947,-179.350,8.931,149.557
C03427=1115.255,164.316,-62.970,-179.348,8.934,149.557
C03428=1115.250,164.565,-62.993,-179.346,8.937,149.557
C03429=1115.246,164.815,-63.015,-179.344,8.940,149.557
C03430=1115.241,165.064,-63.039,-179.341,8.943,149.557
C03431=1115.236,165.313,-63.062,-179.339,8.946,149.557
C03432=1115.232,165.561,-63.084,-179.337,8.949,149.557
C03433=1115.227,165.810,-63.108,-179.335,8.952,149.557
C03434=1115.222,166.059,-63.131,-179.333,8.955,149.557
C03435=1115.218,166.308,-63.153,-179.330,8.958,149.557
C03436=1115.213,166.557,-63.177,-179.328,8.962,149.558
C03437=1115.208,166.806,-63.200,-179.325,8.965,149.558
C03438=1115.204,167.054,-63.222,-179.324,8.967,149.558
C03439=1115.199,167.303,-63.246,-179.321,8.971,149.558
C03440=1115.195,167.552,-63.269,-179.319,8.974,149.558
C03441=1115.191,167.801,-63.292,-179.316,8.977,149.558
C03442=1115.186,168.050,-63.315,-179.315,8.980,149.558
C03443=1115.181,168.299,-63.339,-179.312,8.983,149.558
C03444=1115.177,168.548,-63.362,-179.310,8.986,149.558
C03445=1115.172,168.796,-63.384,-179.308,8.989,149.559
C03446=1115.167,169.045,-63.408,-179.306,8.992,149.559
C03447=1115.163,169.294,-63.431,-179.303,8.995,149.559
C03448=1115.158,169.543,-63.454,-179.301,8.998,149.559
C03449=1115.154,169.792,-63.477,-179.299,9.001,149.559
C03450=1115.149,170.041,-63.501,-179.297,9.004,149.559
C03451=1115.144,170.290,-63.524,-179.295,9.007,149.559
C03452=1115.140,170.539,-63.547,-179.292,9.010,149.559
C03453=1115.135,170.788,-63.571,-179.290,9.013,149.559
C03454=1115.131,171.002,-63.590,-179.288,9.016,149.560
C03455=1115.128,171.215,-63.610,-179.286,9.018,149.560
C03456=1115.124,171.429,-63.630,-179.285,9.021,149.560
C03457=1115.119,171.643,-63.650,-179.283,9.023,149.560
C03458=1115.115,171.856,-63.670,-179.281,9.026,149.560
C03459=1115.112,172.069,-63.691,-179.279,9.029,149.560
C03460=1115.107,172.283,-63.711,-179.277,9.031,149.560
C03461=1115.104,172.497,-63.731,-179.275,9.034,149.560
C03462=1115.099,172.746,-63.754,-179.273,9.037,149.560
C03463=1115.094,172.995,-63.778,-179.271,9.039,149.560
C03464=1115.090,173.243,-63.800,-179.268,9.043,149.560
C03465=1115.086,173.492,-63.824,-179.266,9.046,149.561
C03466=1115.081,173.741,-63.848,-179.264,9.048,149.561
C03467=1115.077,173.990,-63.871,-179.262,9.051,149.561
C03468=1115.072,174.239,-63.895,-179.260,9.055,149.561
C03469=1115.067,174.487,-63.919,-179.258,9.057,149.561
C03470=1115.063,174.736,-63.942,-179.255,9.060,149.561
C03471=1115.058,174.985,-63.965,-179.253,9.064,149.561
C03472=1115.053,175.234,-63.989,-179.251,9.066,149.561
C03473=1115.049,175.483,-64.013,-179.249,9.069,149.561
C03474=1115.044,175.732,-64.036,-179.247,9.073,149.561
C03475=1115.040,175.981,-64.060,-179.245,9.075,149.561
C03476=1115.035,176.229,-64.084,-179.242,9.078,149.562
C03477=1115.030,176.478,-64.107,-179.240,9.082,149.562
C03478=1115.026,176.727,-64.130,-179.238,9.084,149.562
C03479=1115.021,176.976,-64.154,-179.236,9.087,149.562
C03480=1115.017,177.225,-64.178,-179.234,9.091,149.562
C03481=1115.013,177.474,-64.202,-179.232,9.093,149.562
C03482=1115.008,177.723,-64.226,-179.229,9.096,149.562
C03483=1115.003,177.972,-64.249,-179.227,9.099,149.562
C03484=1114.999,178.220,-64.273,-179.225,9.102,149.562
C03485=1114.994,178.469,-64.296,-179.223,9.105,149.562
C03486=1114.990,178.718,-64.320,-179.221,9.108,149.563
C03487=1114.985,178.967,-64.344,-179.219,9.111,149.563
C03488=1114.981,179.215,-64.368,-179.216,9.114,149.563
C03489=1114.976,179.464,-64.391,-179.214,9.117,149.563
C03490=1114.972,179.713,-64.415,-179.211,9.120,149.563
C03491=1114.967,179.962,-64.439,-179.209,9.123,149.563
C03492=1114.963,180.211,-64.463,-179.206,9.126,149.563
C03493=1114.959,180.460,-64.486,-179.204,9.129,149.563
C03494=1114.954,180.708,-64.510,-179.201,9.133,149.563
C03495=1114.949,180.958,-64.534,-179.199,9.136,149.563
C03496=1114.944,181.206,-64.559,-179.196,9.139,149.563
C03497=1114.940,181.455,-64.583,-179.194,9.142,149.563
C03498=1114.936,181.704,-64.606,-179.191,9.145,149.563
C03499=1114.932,181.953,-64.630,-179.189,9.148,149.563
C03500=1114.927,182.201,-64.654,-179.186,9.151,149.563
C03501=1114.922,182.450,-64.678,-179.184,9.154,149.563
C03502=1114.917,182.699,-64.703,-179.182,9.157,149.563
C03503=1114.913,182.947,-64.727,-179.179,9.160,149.563
C03504=1114.909,183.197,-64.750,-179.177,9.163,149.564
C03505=1114.904,183.445,-64.774,-179.174,9.166,149.564
C03506=1114.899,183.694,-64.799,-179.172,9.169,149.564
C03507=1114.895,183.943,-64.822,-179.169,9.172,149.564
C03508=1114.890,184.192,-64.846,-179.167,9.175,149.564
C03509=1114.886,184.441,-64.871,-179.165,9.178,149.564
C03510=1114.882,184.655,-64.891,-179.162,9.181,149.564
C03511=1114.878,184.867,-64.912,-179.160,9.183,149.564
C03512=1114.874,185.081,-64.933,-179.158,9.185,149.564
C03513=1114.870,185.295,-64.954,-179.156,9.188,149.564
C03514=1114.867,185.508,-64.974,-179.153,9.190,149.564
C03515=1114.863,185.722,-64.995,-179.152,9.193,149.564
C03516=1114.858,185.935,-65.016,-179.150,9.195,149.564
C03517=1114.855,186.149,-65.037,-179.148,9.197,149.564
C03518=1114.850,186.398,-65.061,-179.145,9.201,149.564
C03519=1114.846,186.646,-65.085,-179.143,9.204,149.564
C03520=1114.841,186.895,-65.109,-179.141,9.206,149.564
C03521=1114.837,187.144,-65.134,-179.138,9.209,149.564
C03522=1114.832,187.392,-65.159,-179.136,9.212,149.564
C03523=1114.828,187.641,-65.182,-179.134,9.215,149.564
C03524=1114.823,187.890,-65.207,-179.131,9.218,149.564
C03525=1114.819,188.139,-65.231,-179.129,9.221,149.564
C03526=1114.814,188.388,-65.255,-179.127,9.223,149.564
C03527=1114.809,188.636,-65.280,-179.124,9.226,149.564
C03528=1114.805,188.886,-65.304,-179.123,9.229,149.564
C03529=1114.800,189.134,-65.329,-179.120,9.232,149.564
C03530=1114.796,189.383,-65.353,-179.118,9.235,149.564
C03531=1114.792,189.632,-65.377,-179.116,9.237,149.564
C03532=1114.787,189.880,-65.402,-179.113,9.240,149.564
C03533=1114.783,190.129,-65.426,-179.111,9.243,149.565
C03534=1114.778,190.378,-65.451,-179.109,9.246,149.565
C03535=1114.774,190.627,-65.475,-179.107,9.248,149.565
C03536=1114.769,190.875,-65.500,-179.104,9.251,149.565
C03537=1114.765,191.125,-65.524,-179.102,9.253,149.565
C03538=1114.760,191.373,-65.549,-179.100,9.257,149.565
C03539=1114.756,191.621,-65.574,-179.098,9.259,149.565
C03540=1114.751,191.871,-65.599,-179.096,9.262,149.565
C03541=1114.747,192.119,-65.623,-179.094,9.265,149.565
C03542=1114.741,192.368,-65.648,-179.091,9.268,149.565
C03543=1114.738,192.617,-65.672,-179.090,9.270,149.565
C03544=1114.733,192.865,-65.697,-179.087,9.273,149.565
C03545=1114.728,193.114,-65.721,-179.085,9.276,149.565
C03546=1114.724,193.363,-65.747,-179.083,9.279,149.565
C03547=1114.720,193.611,-65.771,-179.081,9.281,149.566
C03548=1114.715,193.861,-65.796,-179.079,9.285,149.566
C03549=1114.711,194.109,-65.820,-179.077,9.287,149.566
C03550=1114.705,194.358,-65.844,-179.075,9.290,149.566
C03551=1114.702,194.606,-65.870,-179.073,9.293,149.566
C03552=1114.697,194.855,-65.894,-179.071,9.295,149.566
C03553=1114.692,195.104,-65.919,-179.068,9.298,149.566
C03554=1114.688,195.353,-65.943,-179.067,9.301,149.566
C03555=1114.683,195.601,-65.969,-179.065,9.303,149.566
C03556=1114.679,195.850,-65.993,-179.063,9.307,149.567
C03557=1114.674,196.099,-66.018,-179.061,9.309,149.567
C03558=1114.670,196.348,-66.043,-179.059,9.311,149.567
C03559=1114.666,196.596,-66.068,-179.056,9.315,149.567
C03560=1114.661,196.845,-66.093,-179.053,9.318,149.567
C03561=1114.657,197.094,-66.117,-179.051,9.321,149.567
C03562=1114.652,197.343,-66.142,-179.047,9.325,149.567
C03563=1114.647,197.591,-66.167,-179.045,9.328,149.567
C03564=1114.644,197.840,-66.192,-179.042,9.331,149.567
C03565=1114.639,198.088,-66.217,-179.039,9.335,149.567
C03566=1114.635,198.302,-66.238,-179.037,9.337,149.567
C03567=1114.631,198.516,-66.260,-179.034,9.340,149.567
C03568=1114.627,198.728,-66.281,-179.031,9.343,149.567
C03569=1114.623,198.942,-66.303,-179.029,9.345,149.567
C03570=1114.619,199.156,-66.324,-179.026,9.348,149.566
C03571=1114.616,199.369,-66.345,-179.025,9.350,149.566
C03572=1114.612,199.582,-66.367,-179.022,9.353,149.566
C03573=1114.608,199.796,-66.389,-179.019,9.356,149.566
C03574=1114.603,200.044,-66.414,-179.016,9.359,149.566
C03575=1114.599,200.293,-66.439,-179.014,9.362,149.566
C03576=1114.595,200.541,-66.464,-179.011,9.365,149.566
C03577=1114.590,200.791,-66.489,-179.008,9.368,149.566
C03578=1114.586,201.040,-66.515,-179.005,9.371,149.566
C03579=1114.581,201.288,-66.539,-179.002,9.374,149.566
C03580=1114.577,201.537,-66.565,-178.999,9.377,149.566
C03581=1114.572,201.785,-66.590,-178.996,9.380,149.566
C03582=1114.568,202.034,-66.615,-178.993,9.383,149.566
C03583=1114.563,202.282,-66.640,-178.991,9.386,149.566
C03584=1114.558,202.532,-66.665,-178.988,9.388,149.566
C03585=1114.555,202.780,-66.691,-178.985,9.391,149.565
C03586=1114.550,203.028,-66.716,-178.981,9.395,149.565
C03587=1114.546,203.277,-66.742,-178.979,9.398,149.565
C03588=1114.541,203.526,-66.766,-178.976,9.401,149.565
C03589=1114.537,203.775,-66.792,-178.973,9.403,149.565
C03590=1114.532,204.024,-66.818,-178.970,9.406,149.565
C03591=1114.527,204.272,-66.843,-178.967,9.409,149.565
C03592=1114.523,204.521,-66.868,-178.964,9.412,149.565
C03593=1114.519,204.770,-66.894,-178.961,9.415,149.565
C03594=1114.514,205.018,-66.919,-178.958,9.417,149.565
C03595=1114.510,205.267,-66.945,-178.956,9.421,149.565
C03596=1114.505,205.515,-66.969,-178.953,9.423,149.564
C03597=1114.501,205.764,-66.995,-178.950,9.426,149.564
C03598=1114.497,206.013,-67.021,-178.947,9.429,149.564
C03599=1114.492,206.261,-67.046,-178.944,9.432,149.564
C03600=1114.488,206.510,-67.072,-178.942,9.435,149.564
C03601=1114.484,206.759,-67.098,-178.939,9.437,149.564
C03602=1114.479,207.007,-67.123,-178.935,9.441,149.564
C03603=1114.474,207.256,-67.148,-178.932,9.444,149.564
C03604=1114.470,207.505,-67.174,-178.930,9.447,149.564
C03605=1114.466,207.754,-67.200,-178.927,9.450,149.564
C03606=1114.460,208.002,-67.226,-178.924,9.453,149.564
C03607=1114.456,208.251,-67.251,-178.921,9.455,149.564
C03608=1114.452,208.500,-67.277,-178.919,9.458,149.564
C03609=1114.447,208.748,-67.302,-178.916,9.461,149.563
C03610=1114.443,208.997,-67.328,-178.913,9.464,149.563
C03611=1114.438,209.245,-67.354,-178.910,9.467,149.563
C03612=1114.434,209.494,-67.380,-178.907,9.470,149.563
C03613=1114.429,209.742,-67.405,-178.905,9.473,149.563
C03614=1114.425,209.991,-67.431,-178.902,9.476,149.563
C03615=1114.421,210.239,-67.457,-178.899,9.479,149.563
C03616=1114.417,210.488,-67.483,-178.896,9.481,149.563
C03617=1114.412,210.737,-67.509,-178.894,9.485,149.563
C03618=1114.407,210.985,-67.535,-178.891,9.487,149.563
C03619=1114.403,211.234,-67.561,-178.888,9.490,149.563
C03620=1114.399,211.483,-67.586,-178.886,9.494,149.563
C03621=1114.395,211.732,-67.612,-178.883,9.496,149.563
C03622=1114.390,211.945,-67.634,-178.880,9.499,149.563
C03623=1114.387,212.158,-67.657,-178.878,9.502,149.563
C03624=1114.383,212.371,-67.679,-178.875,9.504,149.563
C03625=1114.379,212.584,-67.701,-178.874,9.507,149.563
C03626=1114.375,212.798,-67.723,-178.871,9.510,149.563
C03627=1114.371,213.011,-67.746,-178.868,9.513,149.563
C03628=1114.368,213.225,-67.768,-178.867,9.515,149.563
C03629=1114.364,213.437,-67.790,-178.864,9.518,149.563
C03630=1114.359,213.686,-67.817,-178.862,9.521,149.563
C03631=1114.355,213.935,-67.842,-178.860,9.524,149.563
C03632=1114.351,214.183,-67.869,-178.858,9.526,149.563
C03633=1114.347,214.432,-67.895,-178.856,9.530,149.564
C03634=1114.342,214.681,-67.921,-178.854,9.532,149.564
C03635=1114.337,214.929,-67.946,-178.851,9.535,149.564
C03636=1114.333,215.178,-67.973,-178.849,9.538,149.564
C03637=1114.329,215.426,-67.999,-178.847,9.541,149.564
C03638=1114.324,215.675,-68.026,-178.845,9.544,149.564
C03639=1114.320,215.924,-68.051,-178.842,9.547,149.564
C03640=1114.316,216.172,-68.077,-178.841,9.550,149.564
C03641=1114.311,216.421,-68.104,-178.838,9.553,149.564
C03642=1114.307,216.670,-68.130,-178.836,9.556,149.565
C03643=1114.303,216.919,-68.156,-178.834,9.558,149.565
C03644=1114.297,217.166,-68.182,-178.832,9.562,149.565
C03645=1114.293,217.415,-68.208,-178.829,9.565,149.565
C03646=1114.289,217.663,-68.235,-178.827,9.568,149.565
C03647=1114.284,217.913,-68.261,-178.825,9.570,149.565
C03648=1114.280,218.161,-68.287,-178.823,9.574,149.565
C03649=1114.276,218.409,-68.313,-178.820,9.577,149.565
C03650=1114.272,218.658,-68.340,-178.818,9.580,149.565
C03651=1114.267,218.907,-68.366,-178.815,9.583,149.566
C03652=1114.263,219.155,-68.393,-178.813,9.586,149.566
C03653=1114.258,219.404,-68.419,-178.811,9.589,149.566
C03654=1114.255,219.652,-68.445,-178.809,9.592,149.566
C03655=1114.250,219.901,-68.472,-178.806,9.595,149.566
C03656=1114.246,220.150,-68.498,-178.803,9.598,149.566
C03657=1114.241,220.398,-68.525,-178.801,9.602,149.566
C03658=1114.237,220.647,-68.551,-178.798,9.605,149.566
